// TIA Portal V20 export
FUNCTION_BLOCK "CallEquipment"   // FB17, LAD
TITLE = CallEquipment
AUTHOR : ERsystem_FA2_DH. Kim
// This block contains the logic and futher calls (e.g. sequences, control modules, diagnostics etc.) of the equipment module.
// stored: IsIECCheckEnabled true, MemoryReserve 100, Namespace Unit1.Em2, SetENOAutomatically false
   VAR_INPUT
      ZoneOperationEnable { ExternalWritable := 'False'} : "LWONIK_typeSafetyZoneManualOperation";
   END_VAR
   VAR_IN_OUT
      unitStatus : "LAF_typeUnitStatus";   // Current unit status o be used in this EM
      unitAlarmDB : "LAF_typeAlarms";   // Summarized EM Alarms for the Unit
      emFeedback : "LUC_typeEmFeedback";   // Feedback of the EM to the Unit
   END_VAR
   VAR
      instSequenceSemiAutoSplice { ExternalWritable := 'False'} : "Unit1.Em2.Sequence_1_SemiAutoSplice";   // EM Sequence Instance
      instHomeJob1 { S7_SetPoint := 'True'} : "LAF_SelectJob";
      instJob2 { S7_SetPoint := 'True'} : "LAF_SelectJob";
      instJob3 { S7_SetPoint := 'True'} : "LAF_SelectJob";
      instJob4 { S7_SetPoint := 'True'} : "LAF_SelectJob";
      instJob5 { S7_SetPoint := 'True'} : "LAF_SelectJob";
      instJob6 { S7_SetPoint := 'True'} : "LAF_SelectJob";
      instJob7 { S7_SetPoint := 'True'} : "LAF_SelectJob";
      instJob8 { S7_SetPoint := 'True'} : "LAF_SelectJob";
      instJob9 { S7_SetPoint := 'True'} : "LAF_SelectJob";
      instJob10 { S7_SetPoint := 'True'} : "LAF_SelectJob";
      instJob11 { S7_SetPoint := 'True'} : "LAF_SelectJob";
      instJob12 { S7_SetPoint := 'True'} : "LAF_SelectJob";
      instJob13 { S7_SetPoint := 'True'} : "LAF_SelectJob";
      instJob14 { S7_SetPoint := 'True'} : "LAF_SelectJob";
      instJob15 { S7_SetPoint := 'True'} : "LAF_SelectJob";
      instJob16 { S7_SetPoint := 'True'} : "LAF_SelectJob";
      instJob17 { S7_SetPoint := 'True'} : "LAF_SelectJob";
      instJob18 { S7_SetPoint := 'True'} : "LAF_SelectJob";
      instJob19 { S7_SetPoint := 'True'} : "LAF_SelectJob";
      instJob20 { S7_SetPoint := 'True'} : "LAF_SelectJob";
      instJob21 { S7_SetPoint := 'True'} : "LAF_SelectJob";
      instJob22 { S7_SetPoint := 'True'} : "LAF_SelectJob";
      instJob23 { S7_SetPoint := 'True'} : "LAF_SelectJob";
      instJob24 { S7_SetPoint := 'True'} : "LAF_SelectJob";
      instJob25 { S7_SetPoint := 'True'} : "LAF_SelectJob";
      instJob26 { S7_SetPoint := 'True'} : "LAF_SelectJob";
      instJob27 { S7_SetPoint := 'True'} : "LAF_SelectJob";
      instJob28 { S7_SetPoint := 'True'} : "LAF_SelectJob";
      instJob29 { S7_SetPoint := 'True'} : "LAF_SelectJob";
      instJob30 { S7_SetPoint := 'True'} : "LAF_SelectJob";
      instcmSuctionPadTopUpDown { ExternalAccessible := 'False'; ExternalVisible := 'False'; ExternalWritable := 'False'; S7_SetPoint := 'True'} : "LBC_TwoWayActuatorCn";
      instcmSuctionPadBtmUpDown { ExternalAccessible := 'False'; ExternalVisible := 'False'; ExternalWritable := 'False'; S7_SetPoint := 'True'} : "LBC_TwoWayActuatorCn";
      instcmCutterUpDown { ExternalAccessible := 'False'; ExternalVisible := 'False'; ExternalWritable := 'False'; S7_SetPoint := 'True'} : "LBC_TwoWayActuatorCn";
      instcmTapeTopUpDown { ExternalAccessible := 'False'; ExternalVisible := 'False'; ExternalWritable := 'False'; S7_SetPoint := 'True'} : "LBC_TwoWayActuatorCn";
      instcmTapeBtmUpDown { ExternalAccessible := 'False'; ExternalVisible := 'False'; ExternalWritable := 'False'; S7_SetPoint := 'True'} : "LBC_TwoWayActuatorCn";
      instcmSpliceHeadRotateTopFwdBwd { ExternalAccessible := 'False'; ExternalVisible := 'False'; ExternalWritable := 'False'; S7_SetPoint := 'True'} : "LBC_TwoWayActuatorCn";
      instcmSpliceHeadRotateBtmFwdBwd { ExternalAccessible := 'False'; ExternalVisible := 'False'; ExternalWritable := 'False'; S7_SetPoint := 'True'} : "LBC_TwoWayActuatorCn";
      instcmSuctionPadTopLeftVaccum { ExternalAccessible := 'False'; ExternalVisible := 'False'; ExternalWritable := 'False'; S7_SetPoint := 'True'} : "LBC_TwoWayActuatorCn";
      instcmSuctionPadTopRightVaccum { ExternalAccessible := 'False'; ExternalVisible := 'False'; ExternalWritable := 'False'; S7_SetPoint := 'True'} : "LBC_TwoWayActuatorCn";
      instCmSuctionPadBtmLeftVaccum { ExternalAccessible := 'False'; ExternalVisible := 'False'; ExternalWritable := 'False'; S7_SetPoint := 'True'} : "LBC_TwoWayActuatorCn";
      instCmSuctionPadBtmRightVaccum { ExternalAccessible := 'False'; ExternalVisible := 'False'; ExternalWritable := 'False'; S7_SetPoint := 'True'} : "LBC_TwoWayActuatorCn";
      instCmSuctionPadTopTapeVaccum { ExternalAccessible := 'False'; ExternalVisible := 'False'; ExternalWritable := 'False'; S7_SetPoint := 'True'} : "LBC_TwoWayActuatorCn";
      instCmSuctionPadBtmTapeVaccum { ExternalAccessible := 'False'; ExternalVisible := 'False'; ExternalWritable := 'False'; S7_SetPoint := 'True'} : "LBC_TwoWayActuatorCn";
      instManageAlarms { ExternalWritable := 'False'} : "LAF_ManageAlarms";
      instEventsPFE : "Unit1.Em2.EventsPFE";
      statTonTime { ExternalAccessible := 'False'; ExternalVisible := 'False'; ExternalWritable := 'False'} : Array[0..1999] of TON_TIME;
      statTofTime { ExternalAccessible := 'False'; ExternalVisible := 'False'; ExternalWritable := 'False'} : Array[0..99] of TOF_TIME;
      statPulse { ExternalAccessible := 'False'; ExternalVisible := 'False'; ExternalWritable := 'False'} : Array[0..999] of Bool;
      statUnitStatus { ExternalWritable := 'False'} : "LAF_typeUnitStatus";   // Unit Status used in this EM
      statEnableManualCmds : Bool;
      Scan_on { ExternalAccessible := 'False'; ExternalVisible := 'False'; ExternalWritable := 'False'} : Bool;
      "*** Interlock Actuator ******" { ExternalAccessible := 'False'; ExternalVisible := 'False'; ExternalWritable := 'False'; S7_SetPoint := 'True'} : Bool;
      "SuctionPadTopUpDown Home" { S7_SetPoint := 'True'} : "Cylinder.LER_Actuator";
      "SuctionPadTopUpDown Work" { S7_SetPoint := 'True'} : "Cylinder.LER_Actuator";
      "SuctionPadBtmUpDown Home" { S7_SetPoint := 'True'} : "Cylinder.LER_Actuator";
      "SuctionPadBtmUpDown Work" { S7_SetPoint := 'True'} : "Cylinder.LER_Actuator";
      "CutterUpDown Home" { S7_SetPoint := 'True'} : "Cylinder.LER_Actuator";
      "CutterUpDown Work" { S7_SetPoint := 'True'} : "Cylinder.LER_Actuator";
      "TapeTopUpDown Home" { S7_SetPoint := 'True'} : "Cylinder.LER_Actuator";
      "TapeTopUpDown Work" { S7_SetPoint := 'True'} : "Cylinder.LER_Actuator";
      "TapeBtmUpDown Home" { S7_SetPoint := 'True'} : "Cylinder.LER_Actuator";
      "TapeBtmUpDown Work" { S7_SetPoint := 'True'} : "Cylinder.LER_Actuator";
      "SpliceHeadRotateTopFwdBwd Home" { S7_SetPoint := 'True'} : "Cylinder.LER_Actuator";
      "SpliceHeadRotateTopFwdBwd Work" { S7_SetPoint := 'True'} : "Cylinder.LER_Actuator";
      "SpliceHeadRotateBtmFwdBwd Home" { S7_SetPoint := 'True'} : "Cylinder.LER_Actuator";
      "SpliceHeadRotateBtmFwdBwd Work" { S7_SetPoint := 'True'} : "Cylinder.LER_Actuator";
      Cylinder3 : "LER_CM_Name";
      Vaccum1 : "LER_CM_Name";
      Vaccum6 : "LER_CM_Name";
      Cylinder8 : "LER_CM_Name";
      citi_Ptrig : Array[0..20] of Bool;
      citiTon : Array[0..20] of TON_TIME;
      citi : Time;
      citiTest : Array[0..20] of Bool;
   END_VAR
   VAR_TEMP
      tempScInProduction : Bool;   // Mode Production and StateComplete
      tempScNoProduction : Bool;   // Mode Manual and StateComplete
   END_VAR
   VAR CONSTANT
      delayTime : Time := T#3s;
      TRUE : Bool := TRUE;   // Template : Add em specific conditions here
      FALSE : Bool := FALSE;
      NO_JOB : DInt;   // No job
      MIN_POSITION_NUMBER : SInt;
      INIT_POSITION_NUMBER : SInt := -1;
   END_VAR
   VAR_TEMP   // added for the SCL form of the ladder/FBD networks
      _w1 : Bool;
      _w2 : Bool;
      _w3 : Bool;
      _w4 : Bool;
      _w5 : Bool;
      _w6 : Bool;
      _w7 : Bool;
      _w8 : Bool;
      _w9 : Bool;
      _w10 : Bool;
      _w11 : Bool;
      _w12 : Bool;
      _w13 : Bool;
      _w14 : Bool;
      _w15 : Bool;
      _w16 : Bool;
      _w17 : Bool;
      _w18 : Bool;
      _w19 : Bool;
      _w20 : Bool;
   END_VAR
BEGIN

REGION Network 1: BLOCK INFO HEADER
   // (company) / (C) Copyright (year)
   // ---------------------------------------------------------------------------------
   // Title:                             (Title of this block)
   // Comment/Function: (that is implemented in the block)
   // Library/Family:           (that the source is dedicated to)
   // Author:                        (department / person in charge / contact)
   // Target System:          (test system with FW version)
   // Engineering:              TIA Portal (SW version)
   // Restrictions:               (OB types, etc.)
   // Requirements:           (hardware, technological package, etc.)
   // ---------------------------------------------------------------------------------
   // Change log table:
   // Version          | Date             | Signature      | Expert in charge  | Changes applied ------------------------|----------------------|-------------------------|--------------------------------|-----------------------
   // 001.000.000 | yyyy-mm-dd | 0x00000000 | (name of expert) | First released version
END_REGION

REGION Network 2: DESCRIPTION
   // This is a template block provided by the Automation Framework. It can be used to create an own project.
   // The Block Info Header is prepared to put in your own data.
   // Description of the block could be added here and the docu created by Code2Docu.
END_REGION

REGION Network 3: disableFeedbackHomePos
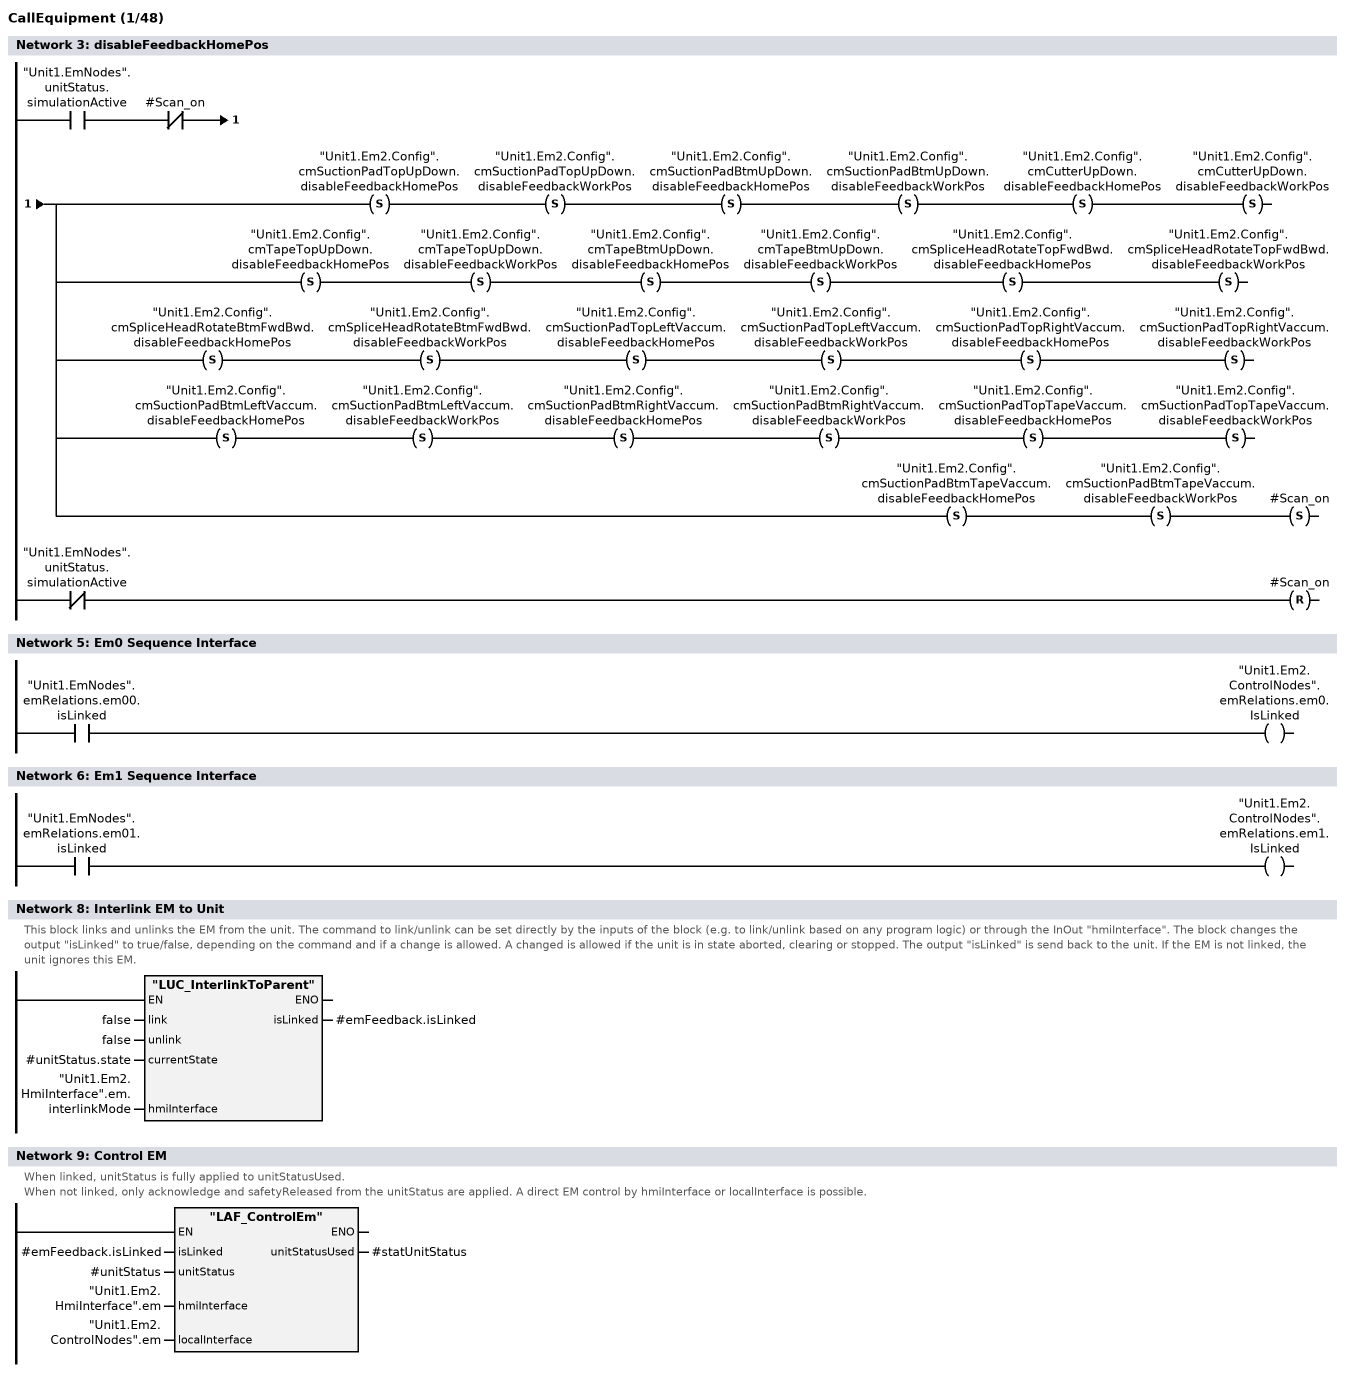
   RUNG wire#powerrail
      Contact( "Unit1.EmNodes".unitStatus.simulationActive )
      I_Contact( #Scan_on )
      wire#w1
      S_Coil( "Unit1.Em2.Config".cmSuctionPadTopUpDown.disableFeedbackHomePos )
      S_Coil( "Unit1.Em2.Config".cmSuctionPadTopUpDown.disableFeedbackWorkPos )
      S_Coil( "Unit1.Em2.Config".cmSuctionPadBtmUpDown.disableFeedbackHomePos )
      S_Coil( "Unit1.Em2.Config".cmSuctionPadBtmUpDown.disableFeedbackWorkPos )
      S_Coil( "Unit1.Em2.Config".cmCutterUpDown.disableFeedbackHomePos )
      S_Coil( "Unit1.Em2.Config".cmCutterUpDown.disableFeedbackWorkPos )
   END_RUNG
   RUNG wire#w1
      S_Coil( "Unit1.Em2.Config".cmTapeTopUpDown.disableFeedbackHomePos )
      S_Coil( "Unit1.Em2.Config".cmTapeTopUpDown.disableFeedbackWorkPos )
      S_Coil( "Unit1.Em2.Config".cmTapeBtmUpDown.disableFeedbackHomePos )
      S_Coil( "Unit1.Em2.Config".cmTapeBtmUpDown.disableFeedbackWorkPos )
      S_Coil( "Unit1.Em2.Config".cmSpliceHeadRotateTopFwdBwd.disableFeedbackHomePos )
      S_Coil( "Unit1.Em2.Config".cmSpliceHeadRotateTopFwdBwd.disableFeedbackWorkPos )
   END_RUNG
   RUNG wire#w1
      S_Coil( "Unit1.Em2.Config".cmSpliceHeadRotateBtmFwdBwd.disableFeedbackHomePos )
      S_Coil( "Unit1.Em2.Config".cmSpliceHeadRotateBtmFwdBwd.disableFeedbackWorkPos )
      S_Coil( "Unit1.Em2.Config".cmSuctionPadTopLeftVaccum.disableFeedbackHomePos )
      S_Coil( "Unit1.Em2.Config".cmSuctionPadTopLeftVaccum.disableFeedbackWorkPos )
      S_Coil( "Unit1.Em2.Config".cmSuctionPadTopRightVaccum.disableFeedbackHomePos )
      S_Coil( "Unit1.Em2.Config".cmSuctionPadTopRightVaccum.disableFeedbackWorkPos )
   END_RUNG
   RUNG wire#w1
      S_Coil( "Unit1.Em2.Config".cmSuctionPadBtmLeftVaccum.disableFeedbackHomePos )
      S_Coil( "Unit1.Em2.Config".cmSuctionPadBtmLeftVaccum.disableFeedbackWorkPos )
      S_Coil( "Unit1.Em2.Config".cmSuctionPadBtmRightVaccum.disableFeedbackHomePos )
      S_Coil( "Unit1.Em2.Config".cmSuctionPadBtmRightVaccum.disableFeedbackWorkPos )
      S_Coil( "Unit1.Em2.Config".cmSuctionPadTopTapeVaccum.disableFeedbackHomePos )
      S_Coil( "Unit1.Em2.Config".cmSuctionPadTopTapeVaccum.disableFeedbackWorkPos )
   END_RUNG
   RUNG wire#w1
      S_Coil( "Unit1.Em2.Config".cmSuctionPadBtmTapeVaccum.disableFeedbackHomePos )
      S_Coil( "Unit1.Em2.Config".cmSuctionPadBtmTapeVaccum.disableFeedbackWorkPos )
      S_Coil( #Scan_on )
   END_RUNG
   RUNG wire#powerrail
      I_Contact( "Unit1.EmNodes".unitStatus.simulationActive )
      R_Coil( #Scan_on )
   END_RUNG
   // the same network as SCL:
   IF "Unit1.EmNodes".unitStatus.simulationActive AND NOT #Scan_on THEN
       "Unit1.Em2.Config".cmSuctionPadTopUpDown.disableFeedbackHomePos := TRUE;
       "Unit1.Em2.Config".cmSuctionPadTopUpDown.disableFeedbackWorkPos := TRUE;
       "Unit1.Em2.Config".cmSuctionPadBtmUpDown.disableFeedbackHomePos := TRUE;
       "Unit1.Em2.Config".cmSuctionPadBtmUpDown.disableFeedbackWorkPos := TRUE;
       "Unit1.Em2.Config".cmCutterUpDown.disableFeedbackHomePos := TRUE;
       "Unit1.Em2.Config".cmCutterUpDown.disableFeedbackWorkPos := TRUE;
       "Unit1.Em2.Config".cmTapeTopUpDown.disableFeedbackHomePos := TRUE;
       "Unit1.Em2.Config".cmTapeTopUpDown.disableFeedbackWorkPos := TRUE;
       "Unit1.Em2.Config".cmTapeBtmUpDown.disableFeedbackHomePos := TRUE;
       "Unit1.Em2.Config".cmTapeBtmUpDown.disableFeedbackWorkPos := TRUE;
       "Unit1.Em2.Config".cmSpliceHeadRotateTopFwdBwd.disableFeedbackHomePos := TRUE;
       "Unit1.Em2.Config".cmSpliceHeadRotateTopFwdBwd.disableFeedbackWorkPos := TRUE;
       "Unit1.Em2.Config".cmSpliceHeadRotateBtmFwdBwd.disableFeedbackHomePos := TRUE;
       "Unit1.Em2.Config".cmSpliceHeadRotateBtmFwdBwd.disableFeedbackWorkPos := TRUE;
       "Unit1.Em2.Config".cmSuctionPadTopLeftVaccum.disableFeedbackHomePos := TRUE;
       "Unit1.Em2.Config".cmSuctionPadTopLeftVaccum.disableFeedbackWorkPos := TRUE;
       "Unit1.Em2.Config".cmSuctionPadTopRightVaccum.disableFeedbackHomePos := TRUE;
       "Unit1.Em2.Config".cmSuctionPadTopRightVaccum.disableFeedbackWorkPos := TRUE;
       "Unit1.Em2.Config".cmSuctionPadBtmLeftVaccum.disableFeedbackHomePos := TRUE;
       "Unit1.Em2.Config".cmSuctionPadBtmLeftVaccum.disableFeedbackWorkPos := TRUE;
       "Unit1.Em2.Config".cmSuctionPadBtmRightVaccum.disableFeedbackHomePos := TRUE;
       "Unit1.Em2.Config".cmSuctionPadBtmRightVaccum.disableFeedbackWorkPos := TRUE;
       "Unit1.Em2.Config".cmSuctionPadTopTapeVaccum.disableFeedbackHomePos := TRUE;
       "Unit1.Em2.Config".cmSuctionPadTopTapeVaccum.disableFeedbackWorkPos := TRUE;
       "Unit1.Em2.Config".cmSuctionPadBtmTapeVaccum.disableFeedbackHomePos := TRUE;
       "Unit1.Em2.Config".cmSuctionPadBtmTapeVaccum.disableFeedbackWorkPos := TRUE;
       #Scan_on := TRUE;
   END_IF;
   IF NOT "Unit1.EmNodes".unitStatus.simulationActive THEN #Scan_on := FALSE; END_IF;
END_REGION

REGION Network 4: ******************** Unit Input ********************
END_REGION

REGION Network 5: Em0 Sequence Interface
   RUNG wire#powerrail
      Contact( "Unit1.EmNodes".emRelations.em00.isLinked )
      Coil( "Unit1.Em2.ControlNodes".emRelations.em0.IsLinked )
   END_RUNG
   // the same network as SCL:
   "Unit1.Em2.ControlNodes".emRelations.em0.IsLinked := "Unit1.EmNodes".emRelations.em00.isLinked;
END_REGION

REGION Network 6: Em1 Sequence Interface
   RUNG wire#powerrail
      Contact( "Unit1.EmNodes".emRelations.em01.isLinked )
      Coil( "Unit1.Em2.ControlNodes".emRelations.em1.IsLinked )
   END_RUNG
   // the same network as SCL:
   "Unit1.Em2.ControlNodes".emRelations.em1.IsLinked := "Unit1.EmNodes".emRelations.em01.isLinked;
END_REGION

REGION Network 7: *************** Equipment Control **************************
END_REGION

REGION Network 8: Interlink EM to Unit
   // This block links and unlinks the EM from the unit. The command to link/unlink can be set directly by the inputs of the block (e.g. to link/unlink based on any program logic) or through the InOut "hmiInterface". The block changes the output "isLinked" to true/false, depending on the command and if a change is allowed. A changed is allowed if the unit is in state aborted, clearing or stopped. The output "isLinked" is send back to the unit. If the EM is not linked, the unit ignores this EM.
   RUNG wire#powerrail
      "LUC_InterlinkToParent"(link := false, unlink := false, currentState := #unitStatus.state, hmiInterface := "Unit1.Em2.HmiInterface".em.interlinkMode, isLinked => #emFeedback.isLinked)
   END_RUNG
   // the same network as SCL:
   "LUC_InterlinkToParent"(link := false,
                           unlink := false,
                           currentState := #unitStatus.state,
                           hmiInterface := "Unit1.Em2.HmiInterface".em.interlinkMode,
                           isLinked => #emFeedback.isLinked);
END_REGION

REGION Network 9: Control EM
   // When linked, unitStatus is fully applied to unitStatusUsed.
   // When not linked, only acknowledge and safetyReleased from the unitStatus are applied. A direct EM control by hmiInterface or localInterface is possible.
   RUNG wire#powerrail
      "LAF_ControlEm"(isLinked := #emFeedback.isLinked, unitStatus := #unitStatus, hmiInterface := "Unit1.Em2.HmiInterface".em, localInterface := "Unit1.Em2.ControlNodes".em, unitStatusUsed => #statUnitStatus)
   END_RUNG
   // the same network as SCL:
   "LAF_ControlEm"(isLinked := #emFeedback.isLinked,
                   unitStatus := #unitStatus,
                   hmiInterface := "Unit1.Em2.HmiInterface".em,
                   localInterface := "Unit1.Em2.ControlNodes".em,
                   unitStatusUsed => #statUnitStatus);
END_REGION

REGION Network 10: EnableManualCmds
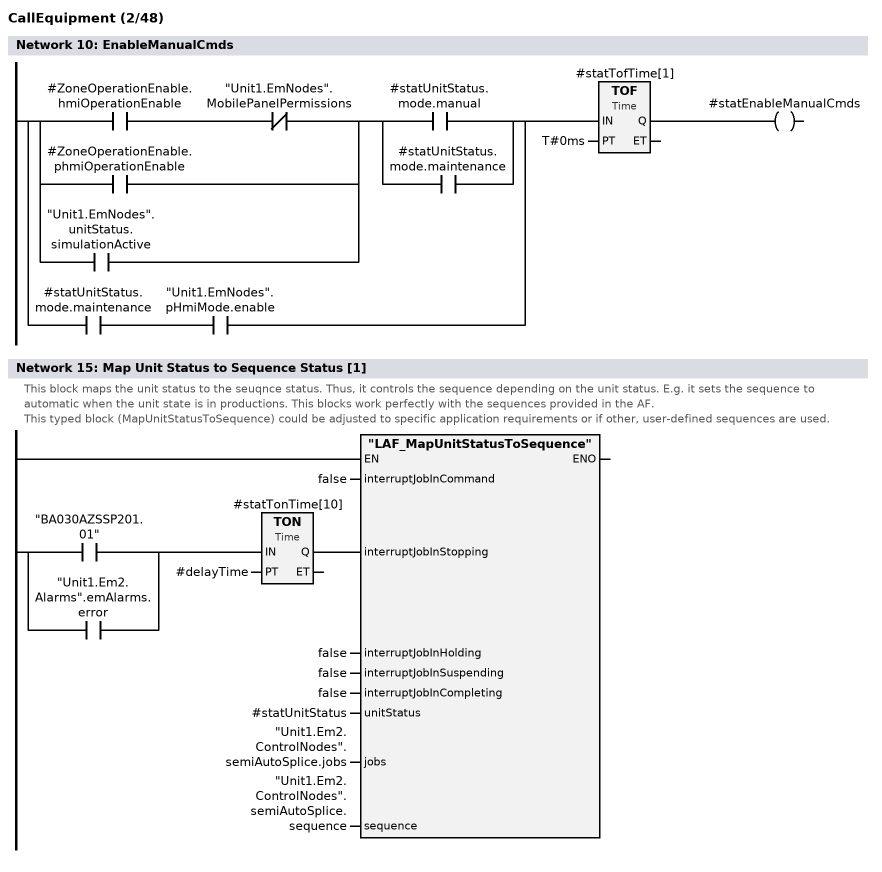
   RUNG wire#powerrail
      Contact( #ZoneOperationEnable.hmiOperationEnable )
      I_Contact( "Unit1.EmNodes".MobilePanelPermissions )
      wire#w1
      Contact( #statUnitStatus.mode.manual )
      wire#w2
      { S7_Templates := "time_type := Time" } #statTofTime[1].TOF(pt := T#0ms, et =>)
      Coil( #statEnableManualCmds )
   END_RUNG
   RUNG wire#powerrail
      Contact( #ZoneOperationEnable.phmiOperationEnable )
   END_RUNG wire#w1
   RUNG wire#powerrail
      Contact( "Unit1.EmNodes".unitStatus.simulationActive )
   END_RUNG wire#w1
   RUNG wire#w1
      Contact( #statUnitStatus.mode.maintenance )
   END_RUNG wire#w2
   RUNG wire#powerrail
      Contact( #statUnitStatus.mode.maintenance )
      Contact( "Unit1.EmNodes".pHmiMode.enable )
   END_RUNG wire#w2
   // the same network as SCL:
   #statTofTime[1].TOF(IN := (((#ZoneOperationEnable.hmiOperationEnable AND NOT "Unit1.EmNodes".MobilePanelPermissions) OR #ZoneOperationEnable.phmiOperationEnable OR "Unit1.EmNodes".unitStatus.simulationActive) AND (#statUnitStatus.mode.manual OR #statUnitStatus.mode.maintenance)) OR (#statUnitStatus.mode.maintenance AND "Unit1.EmNodes".pHmiMode.enable),
                       PT := T#0ms);
   #statEnableManualCmds := #statTofTime[1].Q;
END_REGION

REGION Network 12: *************** Control Modules (Sensors) ********************
   // Call control modules that are sensors before the em logic (jobs and sequence), so that the latest value is used in the logic.
END_REGION

REGION Network 14: *************** Equipment Logic ***************************
END_REGION

REGION Network 15: Map Unit Status to Sequence Status [1]
   // This block maps the unit status to the seuqnce status. Thus, it controls the sequence depending on the unit status. E.g. it sets the sequence to automatic when the unit state is in productions. This blocks work perfectly with the sequences provided in the AF. 
   // This typed block (MapUnitStatusToSequence) could be adjusted to specific application requirements or if other, user-defined sequences are used.
   RUNG wire#powerrail
      "LAF_MapUnitStatusToSequence"(interruptJobInStopping := wire#w2, interruptJobInCommand := false, interruptJobInHolding := false, interruptJobInSuspending := false, interruptJobInCompleting := false, unitStatus := #statUnitStatus, jobs := "Unit1.Em2.ControlNodes".semiAutoSplice.jobs, sequence := "Unit1.Em2.ControlNodes".semiAutoSplice.sequence)
   END_RUNG
   RUNG wire#powerrail
      Contact( "BA030AZSSP201.01" )
      wire#w1
      { S7_Templates := "time_type := Time" } #statTonTime[10].TON(pt := #delayTime, et =>)
   END_RUNG wire#w2
   RUNG wire#powerrail
      Contact( "Unit1.Em2.Alarms".emAlarms.error )
   END_RUNG wire#w1
   // the same network as SCL:
   #statTonTime[10].TON(IN := "BA030AZSSP201.01" OR "Unit1.Em2.Alarms".emAlarms.error, PT := #delayTime);
   "LAF_MapUnitStatusToSequence"(interruptJobInCommand := false,
                           interruptJobInStopping := #statTonTime[10].Q,
                           interruptJobInHolding := false,
                           interruptJobInSuspending := false,
                           interruptJobInCompleting := false,
                           unitStatus := #statUnitStatus,
                           jobs := "Unit1.Em2.ControlNodes".semiAutoSplice.jobs,
                           sequence := "Unit1.Em2.ControlNodes".semiAutoSplice.sequence);
END_REGION

REGION Network 17: Select Job [1] Tape Unit Initialized
   // Decide which Step Sequence to start depending on the OMAC State and EM conditions
   // First Move Block is to Initialize the jobSelect Number
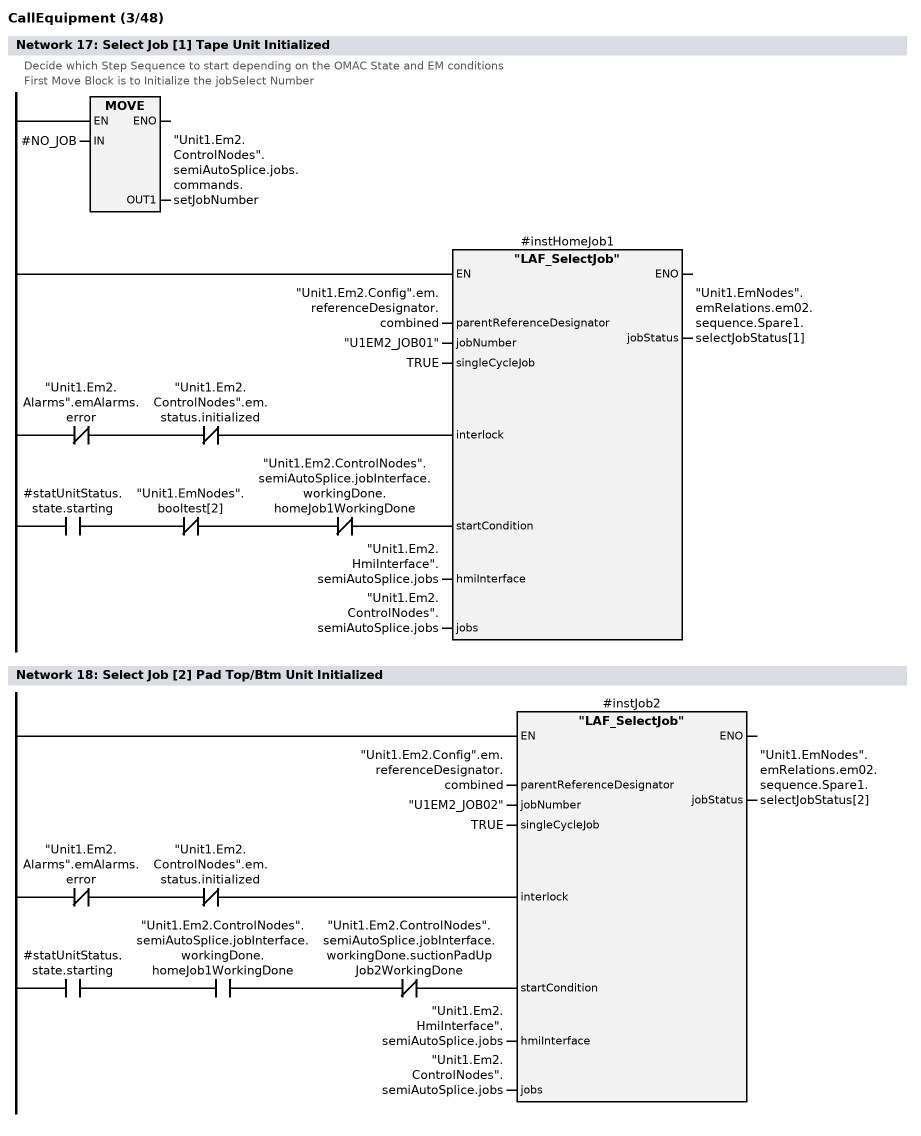
   RUNG wire#powerrail
      Move(in := #NO_JOB, out1 => "Unit1.Em2.ControlNodes".semiAutoSplice.jobs.commands.setJobNumber)
   END_RUNG
   RUNG wire#powerrail
      #instHomeJob1(interlock := wire#w1, startCondition := wire#w2, parentReferenceDesignator := "Unit1.Em2.Config".em.referenceDesignator.combined, jobNumber := "U1EM2_JOB01", singleCycleJob := TRUE, hmiInterface := "Unit1.Em2.HmiInterface".semiAutoSplice.jobs, jobs := "Unit1.Em2.ControlNodes".semiAutoSplice.jobs, jobStatus => "Unit1.EmNodes".emRelations.em02.sequence.Spare1.selectJobStatus[1])
   END_RUNG
   RUNG wire#powerrail
      I_Contact( "Unit1.Em2.Alarms".emAlarms.error )
      I_Contact( "Unit1.Em2.ControlNodes".em.status.initialized )
   END_RUNG wire#w1
   RUNG wire#powerrail
      Contact( #statUnitStatus.state.starting )
      I_Contact( "Unit1.EmNodes".booltest[2] )
      I_Contact( "Unit1.Em2.ControlNodes".semiAutoSplice.jobInterface.workingDone.homeJob1WorkingDone )
   END_RUNG wire#w2
   // the same network as SCL:
   "Unit1.Em2.ControlNodes".semiAutoSplice.jobs.commands.setJobNumber := #NO_JOB;
   #instHomeJob1(parentReferenceDesignator := "Unit1.Em2.Config".em.referenceDesignator.combined,   // "LAF_SelectJob"
                 jobNumber := "U1EM2_JOB01",
                 singleCycleJob := TRUE,
                 interlock := NOT "Unit1.Em2.Alarms".emAlarms.error AND NOT "Unit1.Em2.ControlNodes".em.status.initialized,
                 startCondition := #statUnitStatus.state.starting AND NOT "Unit1.EmNodes".booltest[2] AND NOT "Unit1.Em2.ControlNodes".semiAutoSplice.jobInterface.workingDone.homeJob1WorkingDone,
                 hmiInterface := "Unit1.Em2.HmiInterface".semiAutoSplice.jobs,
                 jobs := "Unit1.Em2.ControlNodes".semiAutoSplice.jobs,
                 jobStatus => "Unit1.EmNodes".emRelations.em02.sequence.Spare1.selectJobStatus[1]);
END_REGION

REGION Network 18: Select Job [2] Pad Top/Btm Unit Initialized
   RUNG wire#powerrail
      #instJob2(interlock := wire#w1, startCondition := wire#w2, parentReferenceDesignator := "Unit1.Em2.Config".em.referenceDesignator.combined, jobNumber := "U1EM2_JOB02", singleCycleJob := TRUE, hmiInterface := "Unit1.Em2.HmiInterface".semiAutoSplice.jobs, jobs := "Unit1.Em2.ControlNodes".semiAutoSplice.jobs, jobStatus => "Unit1.EmNodes".emRelations.em02.sequence.Spare1.selectJobStatus[2])
   END_RUNG
   RUNG wire#powerrail
      I_Contact( "Unit1.Em2.Alarms".emAlarms.error )
      I_Contact( "Unit1.Em2.ControlNodes".em.status.initialized )
   END_RUNG wire#w1
   RUNG wire#powerrail
      Contact( #statUnitStatus.state.starting )
      Contact( "Unit1.Em2.ControlNodes".semiAutoSplice.jobInterface.workingDone.homeJob1WorkingDone )
      I_Contact( "Unit1.Em2.ControlNodes".semiAutoSplice.jobInterface.workingDone.suctionPadUpJob2WorkingDone )
   END_RUNG wire#w2
   // the same network as SCL:
   #instJob2(parentReferenceDesignator := "Unit1.Em2.Config".em.referenceDesignator.combined,   // "LAF_SelectJob"
             jobNumber := "U1EM2_JOB02",
             singleCycleJob := TRUE,
             interlock := NOT "Unit1.Em2.Alarms".emAlarms.error AND NOT "Unit1.Em2.ControlNodes".em.status.initialized,
             startCondition := #statUnitStatus.state.starting AND "Unit1.Em2.ControlNodes".semiAutoSplice.jobInterface.workingDone.homeJob1WorkingDone AND NOT "Unit1.Em2.ControlNodes".semiAutoSplice.jobInterface.workingDone.suctionPadUpJob2WorkingDone,
             hmiInterface := "Unit1.Em2.HmiInterface".semiAutoSplice.jobs,
             jobs := "Unit1.Em2.ControlNodes".semiAutoSplice.jobs,
             jobStatus => "Unit1.EmNodes".emRelations.em02.sequence.Spare1.selectJobStatus[2]);
END_REGION

REGION Network 19: Select Job [3] Head Rotate Top/Btm Unit Initialized
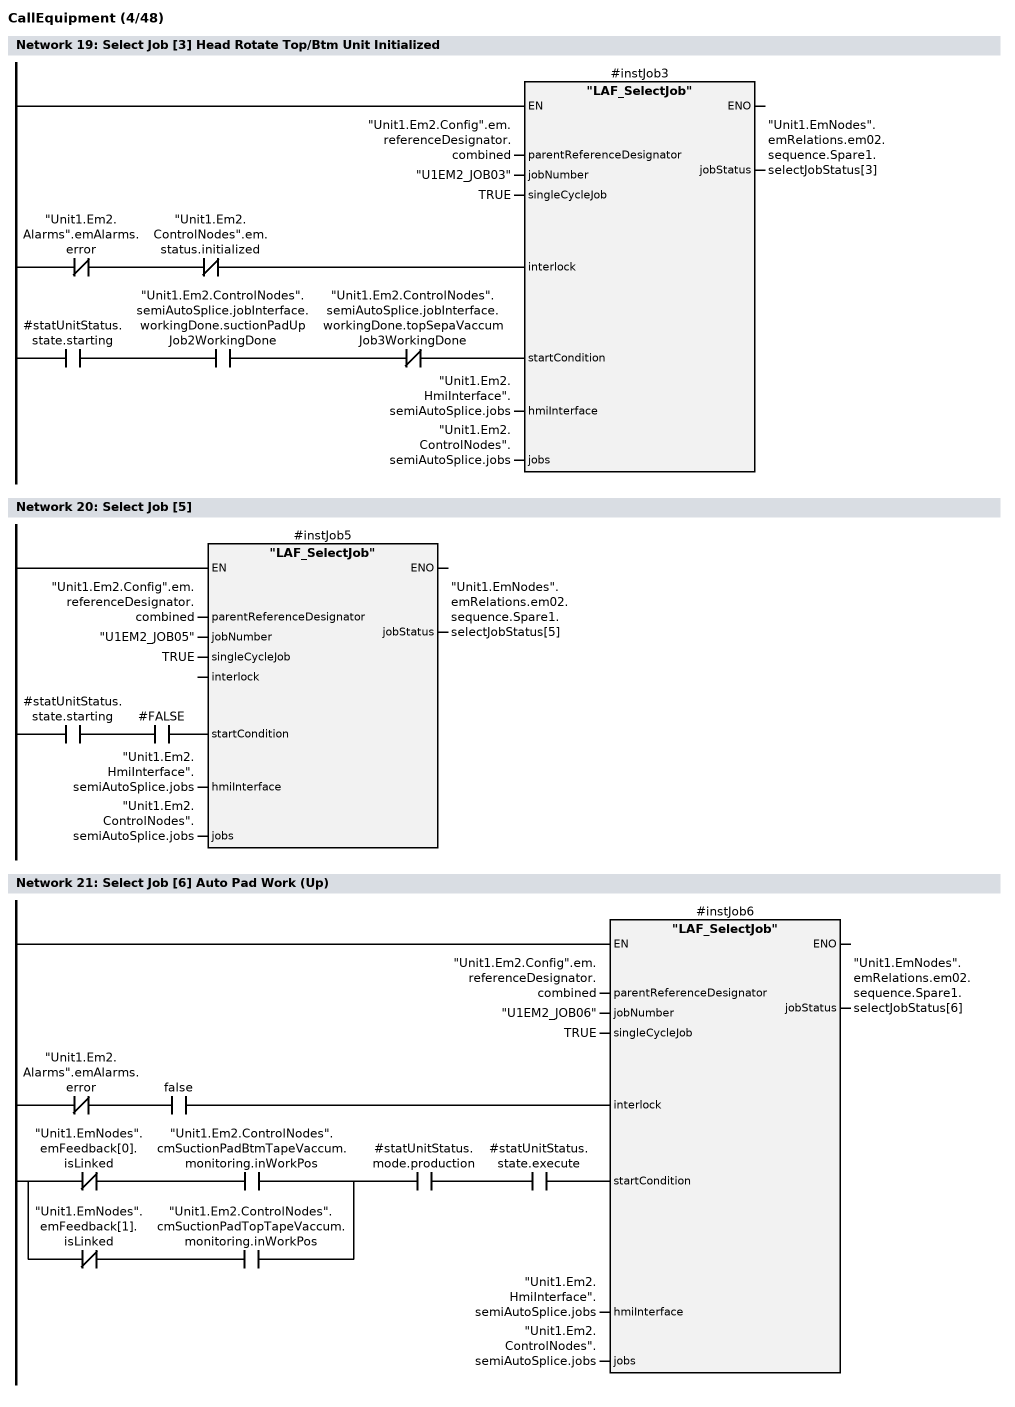
   RUNG wire#powerrail
      #instJob3(interlock := wire#w1, startCondition := wire#w2, parentReferenceDesignator := "Unit1.Em2.Config".em.referenceDesignator.combined, jobNumber := "U1EM2_JOB03", singleCycleJob := TRUE, hmiInterface := "Unit1.Em2.HmiInterface".semiAutoSplice.jobs, jobs := "Unit1.Em2.ControlNodes".semiAutoSplice.jobs, jobStatus => "Unit1.EmNodes".emRelations.em02.sequence.Spare1.selectJobStatus[3])
   END_RUNG
   RUNG wire#powerrail
      I_Contact( "Unit1.Em2.Alarms".emAlarms.error )
      I_Contact( "Unit1.Em2.ControlNodes".em.status.initialized )
   END_RUNG wire#w1
   RUNG wire#powerrail
      Contact( #statUnitStatus.state.starting )
      Contact( "Unit1.Em2.ControlNodes".semiAutoSplice.jobInterface.workingDone.suctionPadUpJob2WorkingDone )
      I_Contact( "Unit1.Em2.ControlNodes".semiAutoSplice.jobInterface.workingDone.topSepaVaccumJob3WorkingDone )
   END_RUNG wire#w2
   // the same network as SCL:
   #instJob3(parentReferenceDesignator := "Unit1.Em2.Config".em.referenceDesignator.combined,   // "LAF_SelectJob"
             jobNumber := "U1EM2_JOB03",
             singleCycleJob := TRUE,
             interlock := NOT "Unit1.Em2.Alarms".emAlarms.error AND NOT "Unit1.Em2.ControlNodes".em.status.initialized,
             startCondition := #statUnitStatus.state.starting AND "Unit1.Em2.ControlNodes".semiAutoSplice.jobInterface.workingDone.suctionPadUpJob2WorkingDone AND NOT "Unit1.Em2.ControlNodes".semiAutoSplice.jobInterface.workingDone.topSepaVaccumJob3WorkingDone,
             hmiInterface := "Unit1.Em2.HmiInterface".semiAutoSplice.jobs,
             jobs := "Unit1.Em2.ControlNodes".semiAutoSplice.jobs,
             jobStatus => "Unit1.EmNodes".emRelations.em02.sequence.Spare1.selectJobStatus[3]);
END_REGION

REGION Network 20: Select Job [5]
   RUNG wire#powerrail
      #instJob5(startCondition := wire#w1, parentReferenceDesignator := "Unit1.Em2.Config".em.referenceDesignator.combined, jobNumber := "U1EM2_JOB05", singleCycleJob := TRUE, interlock :=, hmiInterface := "Unit1.Em2.HmiInterface".semiAutoSplice.jobs, jobs := "Unit1.Em2.ControlNodes".semiAutoSplice.jobs, jobStatus => "Unit1.EmNodes".emRelations.em02.sequence.Spare1.selectJobStatus[5])
   END_RUNG
   RUNG wire#powerrail
      Contact( #statUnitStatus.state.starting )
      Contact( #FALSE )
   END_RUNG wire#w1
   // the same network as SCL:
   #instJob5(parentReferenceDesignator := "Unit1.Em2.Config".em.referenceDesignator.combined,   // "LAF_SelectJob"
             jobNumber := "U1EM2_JOB05",
             singleCycleJob := TRUE,
             startCondition := #statUnitStatus.state.starting AND #FALSE,
             hmiInterface := "Unit1.Em2.HmiInterface".semiAutoSplice.jobs,
             jobs := "Unit1.Em2.ControlNodes".semiAutoSplice.jobs,
             jobStatus => "Unit1.EmNodes".emRelations.em02.sequence.Spare1.selectJobStatus[5]);
END_REGION

REGION Network 21: Select Job [6] Auto Pad Work (Up)
   RUNG wire#powerrail
      #instJob6(interlock := wire#w1, startCondition := wire#w3, parentReferenceDesignator := "Unit1.Em2.Config".em.referenceDesignator.combined, jobNumber := "U1EM2_JOB06", singleCycleJob := TRUE, hmiInterface := "Unit1.Em2.HmiInterface".semiAutoSplice.jobs, jobs := "Unit1.Em2.ControlNodes".semiAutoSplice.jobs, jobStatus => "Unit1.EmNodes".emRelations.em02.sequence.Spare1.selectJobStatus[6])
   END_RUNG
   RUNG wire#powerrail
      I_Contact( "Unit1.Em2.Alarms".emAlarms.error )
      Contact( false )
   END_RUNG wire#w1
   RUNG wire#powerrail
      I_Contact( "Unit1.EmNodes".emFeedback[0].isLinked )
      Contact( "Unit1.Em2.ControlNodes".cmSuctionPadBtmTapeVaccum.monitoring.inWorkPos )
      wire#w2
      Contact( #statUnitStatus.mode.production )
      Contact( #statUnitStatus.state.execute )
   END_RUNG wire#w3
   RUNG wire#powerrail
      I_Contact( "Unit1.EmNodes".emFeedback[1].isLinked )
      Contact( "Unit1.Em2.ControlNodes".cmSuctionPadTopTapeVaccum.monitoring.inWorkPos )
   END_RUNG wire#w2
   // the same network as SCL:
   #instJob6(parentReferenceDesignator := "Unit1.Em2.Config".em.referenceDesignator.combined,   // "LAF_SelectJob"
             jobNumber := "U1EM2_JOB06",
             singleCycleJob := TRUE,
             interlock := NOT "Unit1.Em2.Alarms".emAlarms.error AND false,
             startCondition := ((NOT "Unit1.EmNodes".emFeedback[0].isLinked AND "Unit1.Em2.ControlNodes".cmSuctionPadBtmTapeVaccum.monitoring.inWorkPos) OR (NOT "Unit1.EmNodes".emFeedback[1].isLinked AND "Unit1.Em2.ControlNodes".cmSuctionPadTopTapeVaccum.monitoring.inWorkPos)) AND #statUnitStatus.mode.production AND #statUnitStatus.state.execute,
             hmiInterface := "Unit1.Em2.HmiInterface".semiAutoSplice.jobs,
             jobs := "Unit1.Em2.ControlNodes".semiAutoSplice.jobs,
             jobStatus => "Unit1.EmNodes".emRelations.em02.sequence.Spare1.selectJobStatus[6]);
END_REGION

REGION Network 22: Select Job [7] Auto Suction Pad Vaccum
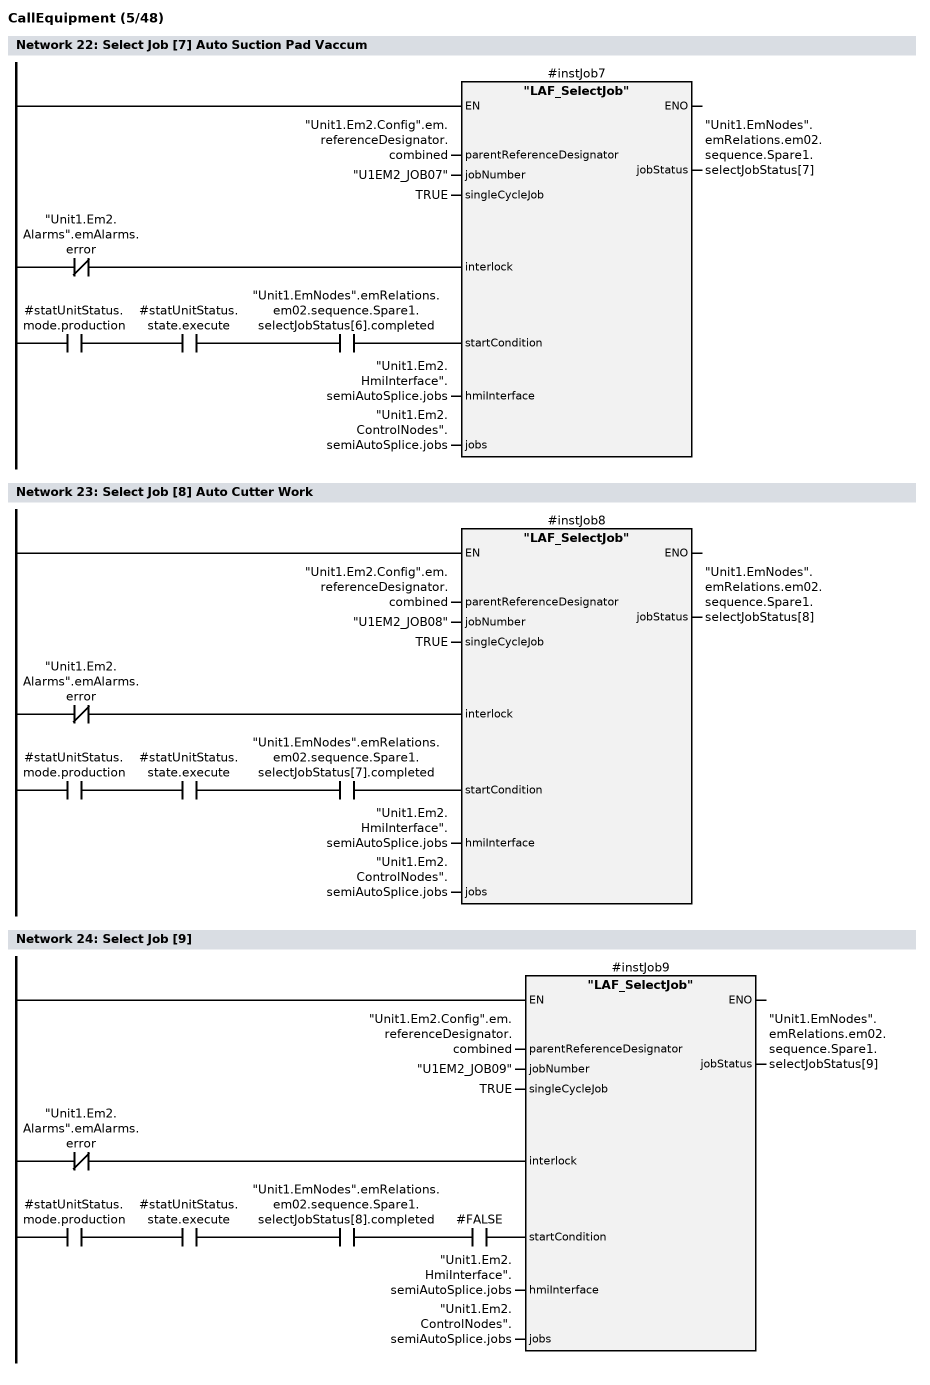
   RUNG wire#powerrail
      #instJob7(interlock := wire#w1, startCondition := wire#w2, parentReferenceDesignator := "Unit1.Em2.Config".em.referenceDesignator.combined, jobNumber := "U1EM2_JOB07", singleCycleJob := TRUE, hmiInterface := "Unit1.Em2.HmiInterface".semiAutoSplice.jobs, jobs := "Unit1.Em2.ControlNodes".semiAutoSplice.jobs, jobStatus => "Unit1.EmNodes".emRelations.em02.sequence.Spare1.selectJobStatus[7])
   END_RUNG
   RUNG wire#powerrail
      I_Contact( "Unit1.Em2.Alarms".emAlarms.error )
   END_RUNG wire#w1
   RUNG wire#powerrail
      Contact( #statUnitStatus.mode.production )
      Contact( #statUnitStatus.state.execute )
      Contact( "Unit1.EmNodes".emRelations.em02.sequence.Spare1.selectJobStatus[6].completed )
   END_RUNG wire#w2
   // the same network as SCL:
   #instJob7(parentReferenceDesignator := "Unit1.Em2.Config".em.referenceDesignator.combined,   // "LAF_SelectJob"
             jobNumber := "U1EM2_JOB07",
             singleCycleJob := TRUE,
             interlock := NOT "Unit1.Em2.Alarms".emAlarms.error,
             startCondition := #statUnitStatus.mode.production AND #statUnitStatus.state.execute AND "Unit1.EmNodes".emRelations.em02.sequence.Spare1.selectJobStatus[6].completed,
             hmiInterface := "Unit1.Em2.HmiInterface".semiAutoSplice.jobs,
             jobs := "Unit1.Em2.ControlNodes".semiAutoSplice.jobs,
             jobStatus => "Unit1.EmNodes".emRelations.em02.sequence.Spare1.selectJobStatus[7]);
END_REGION

REGION Network 23: Select Job [8] Auto Cutter Work
   RUNG wire#powerrail
      #instJob8(interlock := wire#w1, startCondition := wire#w2, parentReferenceDesignator := "Unit1.Em2.Config".em.referenceDesignator.combined, jobNumber := "U1EM2_JOB08", singleCycleJob := TRUE, hmiInterface := "Unit1.Em2.HmiInterface".semiAutoSplice.jobs, jobs := "Unit1.Em2.ControlNodes".semiAutoSplice.jobs, jobStatus => "Unit1.EmNodes".emRelations.em02.sequence.Spare1.selectJobStatus[8])
   END_RUNG
   RUNG wire#powerrail
      I_Contact( "Unit1.Em2.Alarms".emAlarms.error )
   END_RUNG wire#w1
   RUNG wire#powerrail
      Contact( #statUnitStatus.mode.production )
      Contact( #statUnitStatus.state.execute )
      Contact( "Unit1.EmNodes".emRelations.em02.sequence.Spare1.selectJobStatus[7].completed )
   END_RUNG wire#w2
   // the same network as SCL:
   #instJob8(parentReferenceDesignator := "Unit1.Em2.Config".em.referenceDesignator.combined,   // "LAF_SelectJob"
             jobNumber := "U1EM2_JOB08",
             singleCycleJob := TRUE,
             interlock := NOT "Unit1.Em2.Alarms".emAlarms.error,
             startCondition := #statUnitStatus.mode.production AND #statUnitStatus.state.execute AND "Unit1.EmNodes".emRelations.em02.sequence.Spare1.selectJobStatus[7].completed,
             hmiInterface := "Unit1.Em2.HmiInterface".semiAutoSplice.jobs,
             jobs := "Unit1.Em2.ControlNodes".semiAutoSplice.jobs,
             jobStatus => "Unit1.EmNodes".emRelations.em02.sequence.Spare1.selectJobStatus[8]);
END_REGION

REGION Network 24: Select Job [9]
   RUNG wire#powerrail
      #instJob9(interlock := wire#w1, startCondition := wire#w2, parentReferenceDesignator := "Unit1.Em2.Config".em.referenceDesignator.combined, jobNumber := "U1EM2_JOB09", singleCycleJob := TRUE, hmiInterface := "Unit1.Em2.HmiInterface".semiAutoSplice.jobs, jobs := "Unit1.Em2.ControlNodes".semiAutoSplice.jobs, jobStatus => "Unit1.EmNodes".emRelations.em02.sequence.Spare1.selectJobStatus[9])
   END_RUNG
   RUNG wire#powerrail
      I_Contact( "Unit1.Em2.Alarms".emAlarms.error )
   END_RUNG wire#w1
   RUNG wire#powerrail
      Contact( #statUnitStatus.mode.production )
      Contact( #statUnitStatus.state.execute )
      Contact( "Unit1.EmNodes".emRelations.em02.sequence.Spare1.selectJobStatus[8].completed )
      Contact( #FALSE )
   END_RUNG wire#w2
   // the same network as SCL:
   #instJob9(parentReferenceDesignator := "Unit1.Em2.Config".em.referenceDesignator.combined,   // "LAF_SelectJob"
             jobNumber := "U1EM2_JOB09",
             singleCycleJob := TRUE,
             interlock := NOT "Unit1.Em2.Alarms".emAlarms.error,
             startCondition := #statUnitStatus.mode.production AND #statUnitStatus.state.execute AND "Unit1.EmNodes".emRelations.em02.sequence.Spare1.selectJobStatus[8].completed AND #FALSE,
             hmiInterface := "Unit1.Em2.HmiInterface".semiAutoSplice.jobs,
             jobs := "Unit1.Em2.ControlNodes".semiAutoSplice.jobs,
             jobStatus => "Unit1.EmNodes".emRelations.em02.sequence.Spare1.selectJobStatus[9]);
END_REGION

REGION Network 25: Select Job [10] Top to Btm : TOP Vacc Off & Btm Vacc On
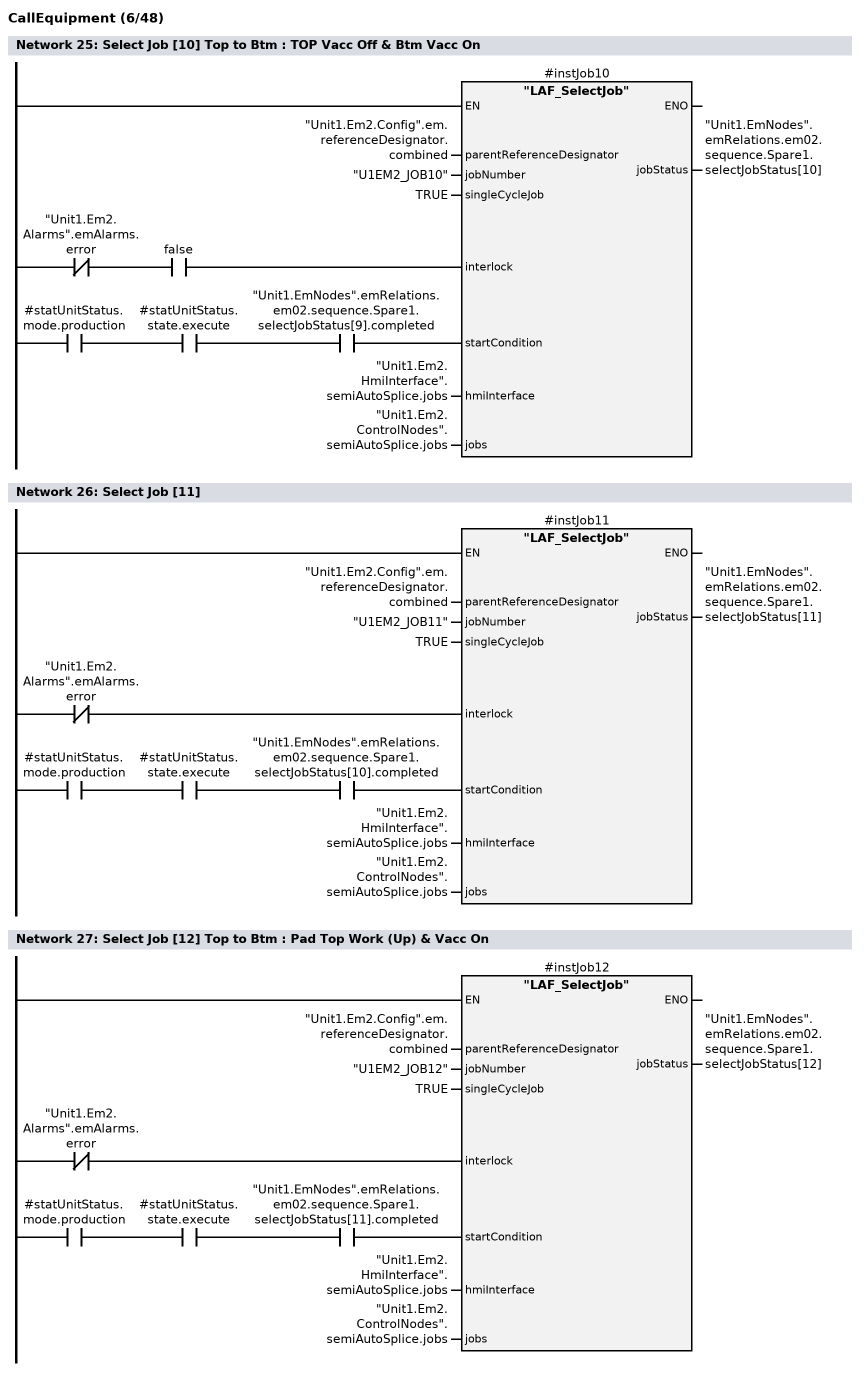
   RUNG wire#powerrail
      #instJob10(interlock := wire#w1, startCondition := wire#w2, parentReferenceDesignator := "Unit1.Em2.Config".em.referenceDesignator.combined, jobNumber := "U1EM2_JOB10", singleCycleJob := TRUE, hmiInterface := "Unit1.Em2.HmiInterface".semiAutoSplice.jobs, jobs := "Unit1.Em2.ControlNodes".semiAutoSplice.jobs, jobStatus => "Unit1.EmNodes".emRelations.em02.sequence.Spare1.selectJobStatus[10])
   END_RUNG
   RUNG wire#powerrail
      I_Contact( "Unit1.Em2.Alarms".emAlarms.error )
      Contact( false )
   END_RUNG wire#w1
   RUNG wire#powerrail
      Contact( #statUnitStatus.mode.production )
      Contact( #statUnitStatus.state.execute )
      Contact( "Unit1.EmNodes".emRelations.em02.sequence.Spare1.selectJobStatus[9].completed )
   END_RUNG wire#w2
   // the same network as SCL:
   #instJob10(parentReferenceDesignator := "Unit1.Em2.Config".em.referenceDesignator.combined,   // "LAF_SelectJob"
              jobNumber := "U1EM2_JOB10",
              singleCycleJob := TRUE,
              interlock := NOT "Unit1.Em2.Alarms".emAlarms.error AND false,
              startCondition := #statUnitStatus.mode.production AND #statUnitStatus.state.execute AND "Unit1.EmNodes".emRelations.em02.sequence.Spare1.selectJobStatus[9].completed,
              hmiInterface := "Unit1.Em2.HmiInterface".semiAutoSplice.jobs,
              jobs := "Unit1.Em2.ControlNodes".semiAutoSplice.jobs,
              jobStatus => "Unit1.EmNodes".emRelations.em02.sequence.Spare1.selectJobStatus[10]);
END_REGION

REGION Network 26: Select Job [11]
   RUNG wire#powerrail
      #instJob11(interlock := wire#w1, startCondition := wire#w2, parentReferenceDesignator := "Unit1.Em2.Config".em.referenceDesignator.combined, jobNumber := "U1EM2_JOB11", singleCycleJob := TRUE, hmiInterface := "Unit1.Em2.HmiInterface".semiAutoSplice.jobs, jobs := "Unit1.Em2.ControlNodes".semiAutoSplice.jobs, jobStatus => "Unit1.EmNodes".emRelations.em02.sequence.Spare1.selectJobStatus[11])
   END_RUNG
   RUNG wire#powerrail
      I_Contact( "Unit1.Em2.Alarms".emAlarms.error )
   END_RUNG wire#w1
   RUNG wire#powerrail
      Contact( #statUnitStatus.mode.production )
      Contact( #statUnitStatus.state.execute )
      Contact( "Unit1.EmNodes".emRelations.em02.sequence.Spare1.selectJobStatus[10].completed )
   END_RUNG wire#w2
   // the same network as SCL:
   #instJob11(parentReferenceDesignator := "Unit1.Em2.Config".em.referenceDesignator.combined,   // "LAF_SelectJob"
              jobNumber := "U1EM2_JOB11",
              singleCycleJob := TRUE,
              interlock := NOT "Unit1.Em2.Alarms".emAlarms.error,
              startCondition := #statUnitStatus.mode.production AND #statUnitStatus.state.execute AND "Unit1.EmNodes".emRelations.em02.sequence.Spare1.selectJobStatus[10].completed,
              hmiInterface := "Unit1.Em2.HmiInterface".semiAutoSplice.jobs,
              jobs := "Unit1.Em2.ControlNodes".semiAutoSplice.jobs,
              jobStatus => "Unit1.EmNodes".emRelations.em02.sequence.Spare1.selectJobStatus[11]);
END_REGION

REGION Network 27: Select Job [12] Top to Btm : Pad Top Work (Up) & Vacc On
   RUNG wire#powerrail
      #instJob12(interlock := wire#w1, startCondition := wire#w2, parentReferenceDesignator := "Unit1.Em2.Config".em.referenceDesignator.combined, jobNumber := "U1EM2_JOB12", singleCycleJob := TRUE, hmiInterface := "Unit1.Em2.HmiInterface".semiAutoSplice.jobs, jobs := "Unit1.Em2.ControlNodes".semiAutoSplice.jobs, jobStatus => "Unit1.EmNodes".emRelations.em02.sequence.Spare1.selectJobStatus[12])
   END_RUNG
   RUNG wire#powerrail
      I_Contact( "Unit1.Em2.Alarms".emAlarms.error )
   END_RUNG wire#w1
   RUNG wire#powerrail
      Contact( #statUnitStatus.mode.production )
      Contact( #statUnitStatus.state.execute )
      Contact( "Unit1.EmNodes".emRelations.em02.sequence.Spare1.selectJobStatus[11].completed )
   END_RUNG wire#w2
   // the same network as SCL:
   #instJob12(parentReferenceDesignator := "Unit1.Em2.Config".em.referenceDesignator.combined,   // "LAF_SelectJob"
              jobNumber := "U1EM2_JOB12",
              singleCycleJob := TRUE,
              interlock := NOT "Unit1.Em2.Alarms".emAlarms.error,
              startCondition := #statUnitStatus.mode.production AND #statUnitStatus.state.execute AND "Unit1.EmNodes".emRelations.em02.sequence.Spare1.selectJobStatus[11].completed,
              hmiInterface := "Unit1.Em2.HmiInterface".semiAutoSplice.jobs,
              jobs := "Unit1.Em2.ControlNodes".semiAutoSplice.jobs,
              jobStatus => "Unit1.EmNodes".emRelations.em02.sequence.Spare1.selectJobStatus[12]);
END_REGION

REGION Network 28: Select Job [13] Top to Btm : BTM Vacc Off & Pad Btm Home (Down)
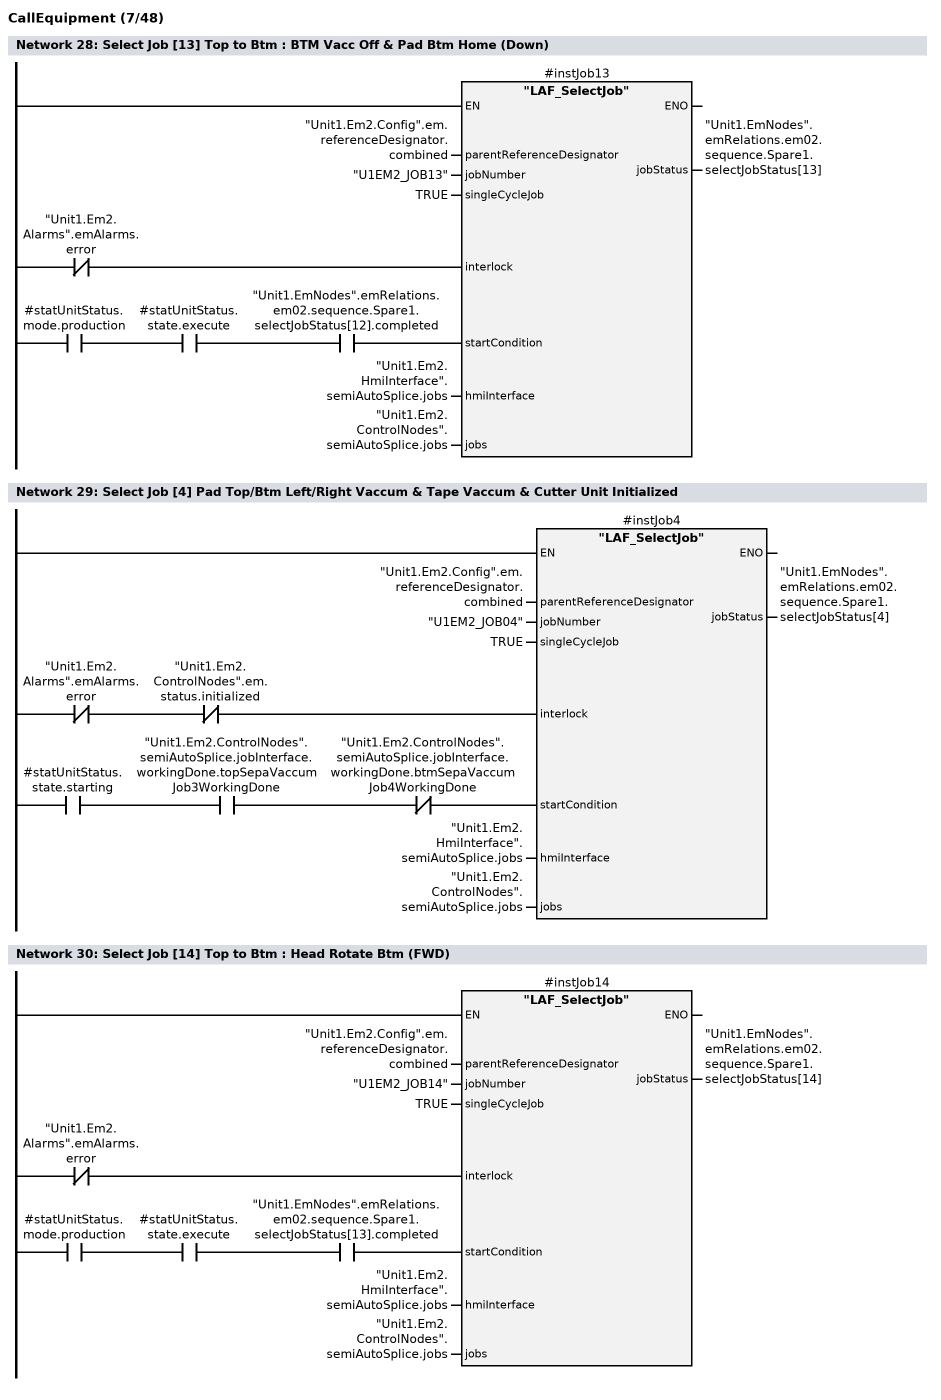
   RUNG wire#powerrail
      #instJob13(interlock := wire#w1, startCondition := wire#w2, parentReferenceDesignator := "Unit1.Em2.Config".em.referenceDesignator.combined, jobNumber := "U1EM2_JOB13", singleCycleJob := TRUE, hmiInterface := "Unit1.Em2.HmiInterface".semiAutoSplice.jobs, jobs := "Unit1.Em2.ControlNodes".semiAutoSplice.jobs, jobStatus => "Unit1.EmNodes".emRelations.em02.sequence.Spare1.selectJobStatus[13])
   END_RUNG
   RUNG wire#powerrail
      I_Contact( "Unit1.Em2.Alarms".emAlarms.error )
   END_RUNG wire#w1
   RUNG wire#powerrail
      Contact( #statUnitStatus.mode.production )
      Contact( #statUnitStatus.state.execute )
      Contact( "Unit1.EmNodes".emRelations.em02.sequence.Spare1.selectJobStatus[12].completed )
   END_RUNG wire#w2
   // the same network as SCL:
   #instJob13(parentReferenceDesignator := "Unit1.Em2.Config".em.referenceDesignator.combined,   // "LAF_SelectJob"
              jobNumber := "U1EM2_JOB13",
              singleCycleJob := TRUE,
              interlock := NOT "Unit1.Em2.Alarms".emAlarms.error,
              startCondition := #statUnitStatus.mode.production AND #statUnitStatus.state.execute AND "Unit1.EmNodes".emRelations.em02.sequence.Spare1.selectJobStatus[12].completed,
              hmiInterface := "Unit1.Em2.HmiInterface".semiAutoSplice.jobs,
              jobs := "Unit1.Em2.ControlNodes".semiAutoSplice.jobs,
              jobStatus => "Unit1.EmNodes".emRelations.em02.sequence.Spare1.selectJobStatus[13]);
END_REGION

REGION Network 29: Select Job [4] Pad Top/Btm Left/Right Vaccum & Tape Vaccum & Cutter Unit Initialized
   RUNG wire#powerrail
      #instJob4(interlock := wire#w1, startCondition := wire#w2, parentReferenceDesignator := "Unit1.Em2.Config".em.referenceDesignator.combined, jobNumber := "U1EM2_JOB04", singleCycleJob := TRUE, hmiInterface := "Unit1.Em2.HmiInterface".semiAutoSplice.jobs, jobs := "Unit1.Em2.ControlNodes".semiAutoSplice.jobs, jobStatus => "Unit1.EmNodes".emRelations.em02.sequence.Spare1.selectJobStatus[4])
   END_RUNG
   RUNG wire#powerrail
      I_Contact( "Unit1.Em2.Alarms".emAlarms.error )
      I_Contact( "Unit1.Em2.ControlNodes".em.status.initialized )
   END_RUNG wire#w1
   RUNG wire#powerrail
      Contact( #statUnitStatus.state.starting )
      Contact( "Unit1.Em2.ControlNodes".semiAutoSplice.jobInterface.workingDone.topSepaVaccumJob3WorkingDone )
      I_Contact( "Unit1.Em2.ControlNodes".semiAutoSplice.jobInterface.workingDone.btmSepaVaccumJob4WorkingDone )
   END_RUNG wire#w2
   // the same network as SCL:
   #instJob4(parentReferenceDesignator := "Unit1.Em2.Config".em.referenceDesignator.combined,   // "LAF_SelectJob"
             jobNumber := "U1EM2_JOB04",
             singleCycleJob := TRUE,
             interlock := NOT "Unit1.Em2.Alarms".emAlarms.error AND NOT "Unit1.Em2.ControlNodes".em.status.initialized,
             startCondition := #statUnitStatus.state.starting AND "Unit1.Em2.ControlNodes".semiAutoSplice.jobInterface.workingDone.topSepaVaccumJob3WorkingDone AND NOT "Unit1.Em2.ControlNodes".semiAutoSplice.jobInterface.workingDone.btmSepaVaccumJob4WorkingDone,
             hmiInterface := "Unit1.Em2.HmiInterface".semiAutoSplice.jobs,
             jobs := "Unit1.Em2.ControlNodes".semiAutoSplice.jobs,
             jobStatus => "Unit1.EmNodes".emRelations.em02.sequence.Spare1.selectJobStatus[4]);
END_REGION

REGION Network 30: Select Job [14] Top to Btm : Head Rotate Btm (FWD)
   RUNG wire#powerrail
      #instJob14(interlock := wire#w1, startCondition := wire#w2, parentReferenceDesignator := "Unit1.Em2.Config".em.referenceDesignator.combined, jobNumber := "U1EM2_JOB14", singleCycleJob := TRUE, hmiInterface := "Unit1.Em2.HmiInterface".semiAutoSplice.jobs, jobs := "Unit1.Em2.ControlNodes".semiAutoSplice.jobs, jobStatus => "Unit1.EmNodes".emRelations.em02.sequence.Spare1.selectJobStatus[14])
   END_RUNG
   RUNG wire#powerrail
      I_Contact( "Unit1.Em2.Alarms".emAlarms.error )
   END_RUNG wire#w1
   RUNG wire#powerrail
      Contact( #statUnitStatus.mode.production )
      Contact( #statUnitStatus.state.execute )
      Contact( "Unit1.EmNodes".emRelations.em02.sequence.Spare1.selectJobStatus[13].completed )
   END_RUNG wire#w2
   // the same network as SCL:
   #instJob14(parentReferenceDesignator := "Unit1.Em2.Config".em.referenceDesignator.combined,   // "LAF_SelectJob"
              jobNumber := "U1EM2_JOB14",
              singleCycleJob := TRUE,
              interlock := NOT "Unit1.Em2.Alarms".emAlarms.error,
              startCondition := #statUnitStatus.mode.production AND #statUnitStatus.state.execute AND "Unit1.EmNodes".emRelations.em02.sequence.Spare1.selectJobStatus[13].completed,
              hmiInterface := "Unit1.Em2.HmiInterface".semiAutoSplice.jobs,
              jobs := "Unit1.Em2.ControlNodes".semiAutoSplice.jobs,
              jobStatus => "Unit1.EmNodes".emRelations.em02.sequence.Spare1.selectJobStatus[14]);
END_REGION

REGION Network 31: Select Job [15] Top to Btm : TAPPING
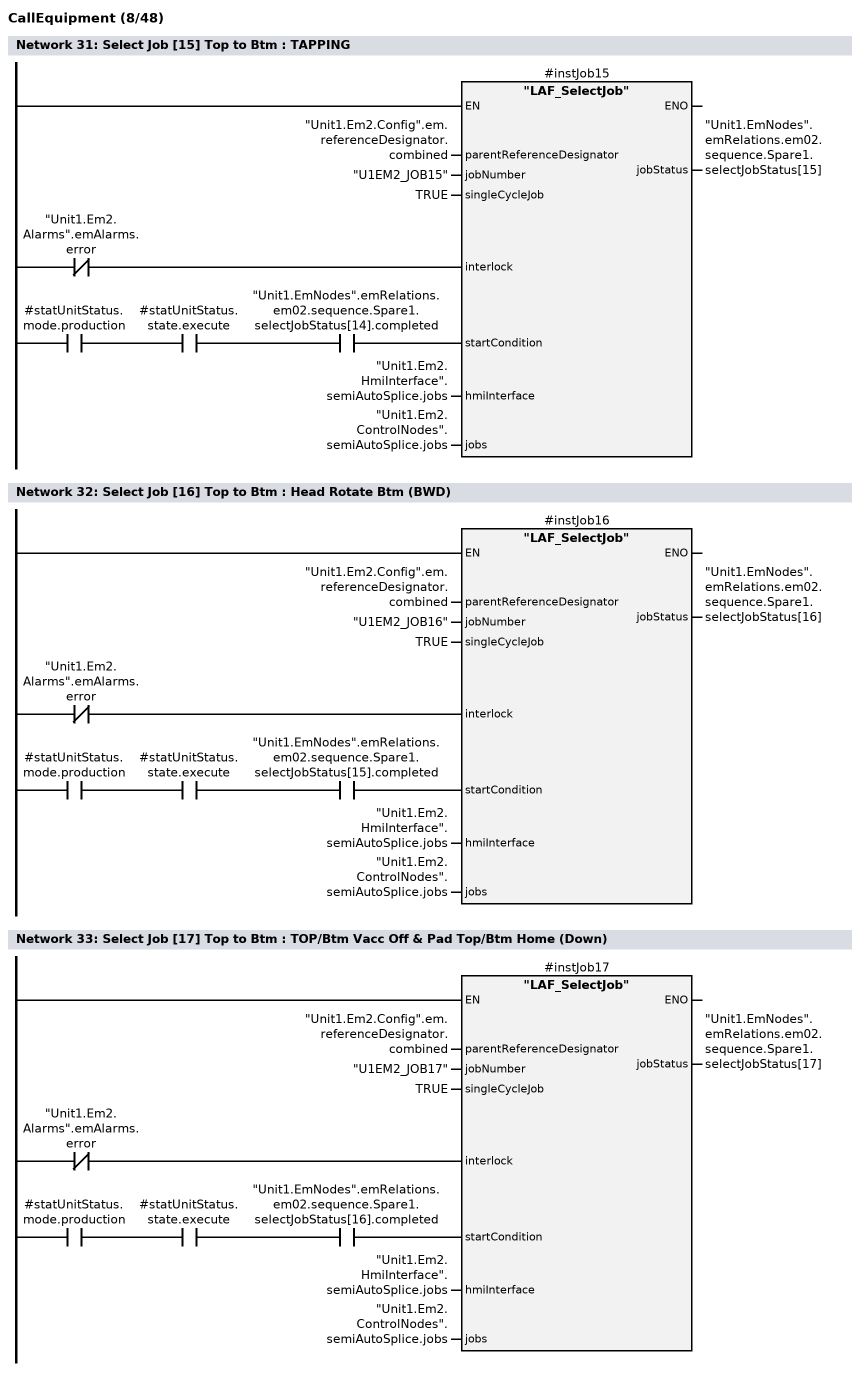
   RUNG wire#powerrail
      #instJob15(interlock := wire#w1, startCondition := wire#w2, parentReferenceDesignator := "Unit1.Em2.Config".em.referenceDesignator.combined, jobNumber := "U1EM2_JOB15", singleCycleJob := TRUE, hmiInterface := "Unit1.Em2.HmiInterface".semiAutoSplice.jobs, jobs := "Unit1.Em2.ControlNodes".semiAutoSplice.jobs, jobStatus => "Unit1.EmNodes".emRelations.em02.sequence.Spare1.selectJobStatus[15])
   END_RUNG
   RUNG wire#powerrail
      I_Contact( "Unit1.Em2.Alarms".emAlarms.error )
   END_RUNG wire#w1
   RUNG wire#powerrail
      Contact( #statUnitStatus.mode.production )
      Contact( #statUnitStatus.state.execute )
      Contact( "Unit1.EmNodes".emRelations.em02.sequence.Spare1.selectJobStatus[14].completed )
   END_RUNG wire#w2
   // the same network as SCL:
   #instJob15(parentReferenceDesignator := "Unit1.Em2.Config".em.referenceDesignator.combined,   // "LAF_SelectJob"
              jobNumber := "U1EM2_JOB15",
              singleCycleJob := TRUE,
              interlock := NOT "Unit1.Em2.Alarms".emAlarms.error,
              startCondition := #statUnitStatus.mode.production AND #statUnitStatus.state.execute AND "Unit1.EmNodes".emRelations.em02.sequence.Spare1.selectJobStatus[14].completed,
              hmiInterface := "Unit1.Em2.HmiInterface".semiAutoSplice.jobs,
              jobs := "Unit1.Em2.ControlNodes".semiAutoSplice.jobs,
              jobStatus => "Unit1.EmNodes".emRelations.em02.sequence.Spare1.selectJobStatus[15]);
END_REGION

REGION Network 32: Select Job [16] Top to Btm : Head Rotate Btm (BWD)
   RUNG wire#powerrail
      #instJob16(interlock := wire#w1, startCondition := wire#w2, parentReferenceDesignator := "Unit1.Em2.Config".em.referenceDesignator.combined, jobNumber := "U1EM2_JOB16", singleCycleJob := TRUE, hmiInterface := "Unit1.Em2.HmiInterface".semiAutoSplice.jobs, jobs := "Unit1.Em2.ControlNodes".semiAutoSplice.jobs, jobStatus => "Unit1.EmNodes".emRelations.em02.sequence.Spare1.selectJobStatus[16])
   END_RUNG
   RUNG wire#powerrail
      I_Contact( "Unit1.Em2.Alarms".emAlarms.error )
   END_RUNG wire#w1
   RUNG wire#powerrail
      Contact( #statUnitStatus.mode.production )
      Contact( #statUnitStatus.state.execute )
      Contact( "Unit1.EmNodes".emRelations.em02.sequence.Spare1.selectJobStatus[15].completed )
   END_RUNG wire#w2
   // the same network as SCL:
   #instJob16(parentReferenceDesignator := "Unit1.Em2.Config".em.referenceDesignator.combined,   // "LAF_SelectJob"
              jobNumber := "U1EM2_JOB16",
              singleCycleJob := TRUE,
              interlock := NOT "Unit1.Em2.Alarms".emAlarms.error,
              startCondition := #statUnitStatus.mode.production AND #statUnitStatus.state.execute AND "Unit1.EmNodes".emRelations.em02.sequence.Spare1.selectJobStatus[15].completed,
              hmiInterface := "Unit1.Em2.HmiInterface".semiAutoSplice.jobs,
              jobs := "Unit1.Em2.ControlNodes".semiAutoSplice.jobs,
              jobStatus => "Unit1.EmNodes".emRelations.em02.sequence.Spare1.selectJobStatus[16]);
END_REGION

REGION Network 33: Select Job [17] Top to Btm : TOP/Btm Vacc Off & Pad Top/Btm Home (Down)
   RUNG wire#powerrail
      #instJob17(interlock := wire#w1, startCondition := wire#w2, parentReferenceDesignator := "Unit1.Em2.Config".em.referenceDesignator.combined, jobNumber := "U1EM2_JOB17", singleCycleJob := TRUE, hmiInterface := "Unit1.Em2.HmiInterface".semiAutoSplice.jobs, jobs := "Unit1.Em2.ControlNodes".semiAutoSplice.jobs, jobStatus => "Unit1.EmNodes".emRelations.em02.sequence.Spare1.selectJobStatus[17])
   END_RUNG
   RUNG wire#powerrail
      I_Contact( "Unit1.Em2.Alarms".emAlarms.error )
   END_RUNG wire#w1
   RUNG wire#powerrail
      Contact( #statUnitStatus.mode.production )
      Contact( #statUnitStatus.state.execute )
      Contact( "Unit1.EmNodes".emRelations.em02.sequence.Spare1.selectJobStatus[16].completed )
   END_RUNG wire#w2
   // the same network as SCL:
   #instJob17(parentReferenceDesignator := "Unit1.Em2.Config".em.referenceDesignator.combined,   // "LAF_SelectJob"
              jobNumber := "U1EM2_JOB17",
              singleCycleJob := TRUE,
              interlock := NOT "Unit1.Em2.Alarms".emAlarms.error,
              startCondition := #statUnitStatus.mode.production AND #statUnitStatus.state.execute AND "Unit1.EmNodes".emRelations.em02.sequence.Spare1.selectJobStatus[16].completed,
              hmiInterface := "Unit1.Em2.HmiInterface".semiAutoSplice.jobs,
              jobs := "Unit1.Em2.ControlNodes".semiAutoSplice.jobs,
              jobStatus => "Unit1.EmNodes".emRelations.em02.sequence.Spare1.selectJobStatus[17]);
END_REGION

REGION Network 34: Select Job [18] Top to Btm : Link Change
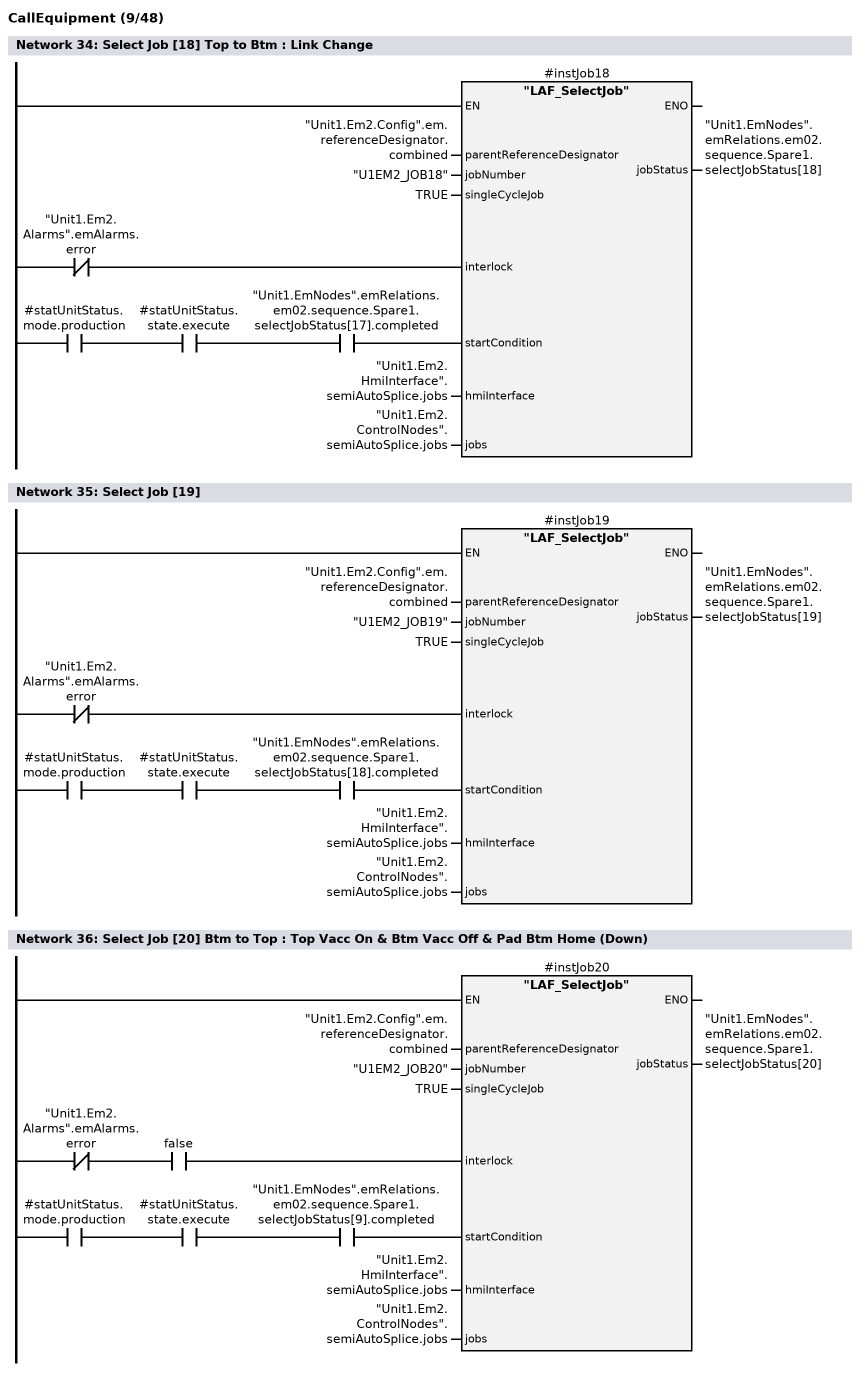
   RUNG wire#powerrail
      #instJob18(interlock := wire#w1, startCondition := wire#w2, parentReferenceDesignator := "Unit1.Em2.Config".em.referenceDesignator.combined, jobNumber := "U1EM2_JOB18", singleCycleJob := TRUE, hmiInterface := "Unit1.Em2.HmiInterface".semiAutoSplice.jobs, jobs := "Unit1.Em2.ControlNodes".semiAutoSplice.jobs, jobStatus => "Unit1.EmNodes".emRelations.em02.sequence.Spare1.selectJobStatus[18])
   END_RUNG
   RUNG wire#powerrail
      I_Contact( "Unit1.Em2.Alarms".emAlarms.error )
   END_RUNG wire#w1
   RUNG wire#powerrail
      Contact( #statUnitStatus.mode.production )
      Contact( #statUnitStatus.state.execute )
      Contact( "Unit1.EmNodes".emRelations.em02.sequence.Spare1.selectJobStatus[17].completed )
   END_RUNG wire#w2
   // the same network as SCL:
   #instJob18(parentReferenceDesignator := "Unit1.Em2.Config".em.referenceDesignator.combined,   // "LAF_SelectJob"
              jobNumber := "U1EM2_JOB18",
              singleCycleJob := TRUE,
              interlock := NOT "Unit1.Em2.Alarms".emAlarms.error,
              startCondition := #statUnitStatus.mode.production AND #statUnitStatus.state.execute AND "Unit1.EmNodes".emRelations.em02.sequence.Spare1.selectJobStatus[17].completed,
              hmiInterface := "Unit1.Em2.HmiInterface".semiAutoSplice.jobs,
              jobs := "Unit1.Em2.ControlNodes".semiAutoSplice.jobs,
              jobStatus => "Unit1.EmNodes".emRelations.em02.sequence.Spare1.selectJobStatus[18]);
END_REGION

REGION Network 35: Select Job [19]
   RUNG wire#powerrail
      #instJob19(interlock := wire#w1, startCondition := wire#w2, parentReferenceDesignator := "Unit1.Em2.Config".em.referenceDesignator.combined, jobNumber := "U1EM2_JOB19", singleCycleJob := TRUE, hmiInterface := "Unit1.Em2.HmiInterface".semiAutoSplice.jobs, jobs := "Unit1.Em2.ControlNodes".semiAutoSplice.jobs, jobStatus => "Unit1.EmNodes".emRelations.em02.sequence.Spare1.selectJobStatus[19])
   END_RUNG
   RUNG wire#powerrail
      I_Contact( "Unit1.Em2.Alarms".emAlarms.error )
   END_RUNG wire#w1
   RUNG wire#powerrail
      Contact( #statUnitStatus.mode.production )
      Contact( #statUnitStatus.state.execute )
      Contact( "Unit1.EmNodes".emRelations.em02.sequence.Spare1.selectJobStatus[18].completed )
   END_RUNG wire#w2
   // the same network as SCL:
   #instJob19(parentReferenceDesignator := "Unit1.Em2.Config".em.referenceDesignator.combined,   // "LAF_SelectJob"
              jobNumber := "U1EM2_JOB19",
              singleCycleJob := TRUE,
              interlock := NOT "Unit1.Em2.Alarms".emAlarms.error,
              startCondition := #statUnitStatus.mode.production AND #statUnitStatus.state.execute AND "Unit1.EmNodes".emRelations.em02.sequence.Spare1.selectJobStatus[18].completed,
              hmiInterface := "Unit1.Em2.HmiInterface".semiAutoSplice.jobs,
              jobs := "Unit1.Em2.ControlNodes".semiAutoSplice.jobs,
              jobStatus => "Unit1.EmNodes".emRelations.em02.sequence.Spare1.selectJobStatus[19]);
END_REGION

REGION Network 36: Select Job [20] Btm to Top : Top Vacc On & Btm Vacc Off & Pad Btm Home (Down)
   RUNG wire#powerrail
      #instJob20(interlock := wire#w1, startCondition := wire#w2, parentReferenceDesignator := "Unit1.Em2.Config".em.referenceDesignator.combined, jobNumber := "U1EM2_JOB20", singleCycleJob := TRUE, hmiInterface := "Unit1.Em2.HmiInterface".semiAutoSplice.jobs, jobs := "Unit1.Em2.ControlNodes".semiAutoSplice.jobs, jobStatus => "Unit1.EmNodes".emRelations.em02.sequence.Spare1.selectJobStatus[20])
   END_RUNG
   RUNG wire#powerrail
      I_Contact( "Unit1.Em2.Alarms".emAlarms.error )
      Contact( false )
   END_RUNG wire#w1
   RUNG wire#powerrail
      Contact( #statUnitStatus.mode.production )
      Contact( #statUnitStatus.state.execute )
      Contact( "Unit1.EmNodes".emRelations.em02.sequence.Spare1.selectJobStatus[9].completed )
   END_RUNG wire#w2
   // the same network as SCL:
   #instJob20(parentReferenceDesignator := "Unit1.Em2.Config".em.referenceDesignator.combined,   // "LAF_SelectJob"
              jobNumber := "U1EM2_JOB20",
              singleCycleJob := TRUE,
              interlock := NOT "Unit1.Em2.Alarms".emAlarms.error AND false,
              startCondition := #statUnitStatus.mode.production AND #statUnitStatus.state.execute AND "Unit1.EmNodes".emRelations.em02.sequence.Spare1.selectJobStatus[9].completed,
              hmiInterface := "Unit1.Em2.HmiInterface".semiAutoSplice.jobs,
              jobs := "Unit1.Em2.ControlNodes".semiAutoSplice.jobs,
              jobStatus => "Unit1.EmNodes".emRelations.em02.sequence.Spare1.selectJobStatus[20]);
END_REGION

REGION Network 37: Select Job [21]
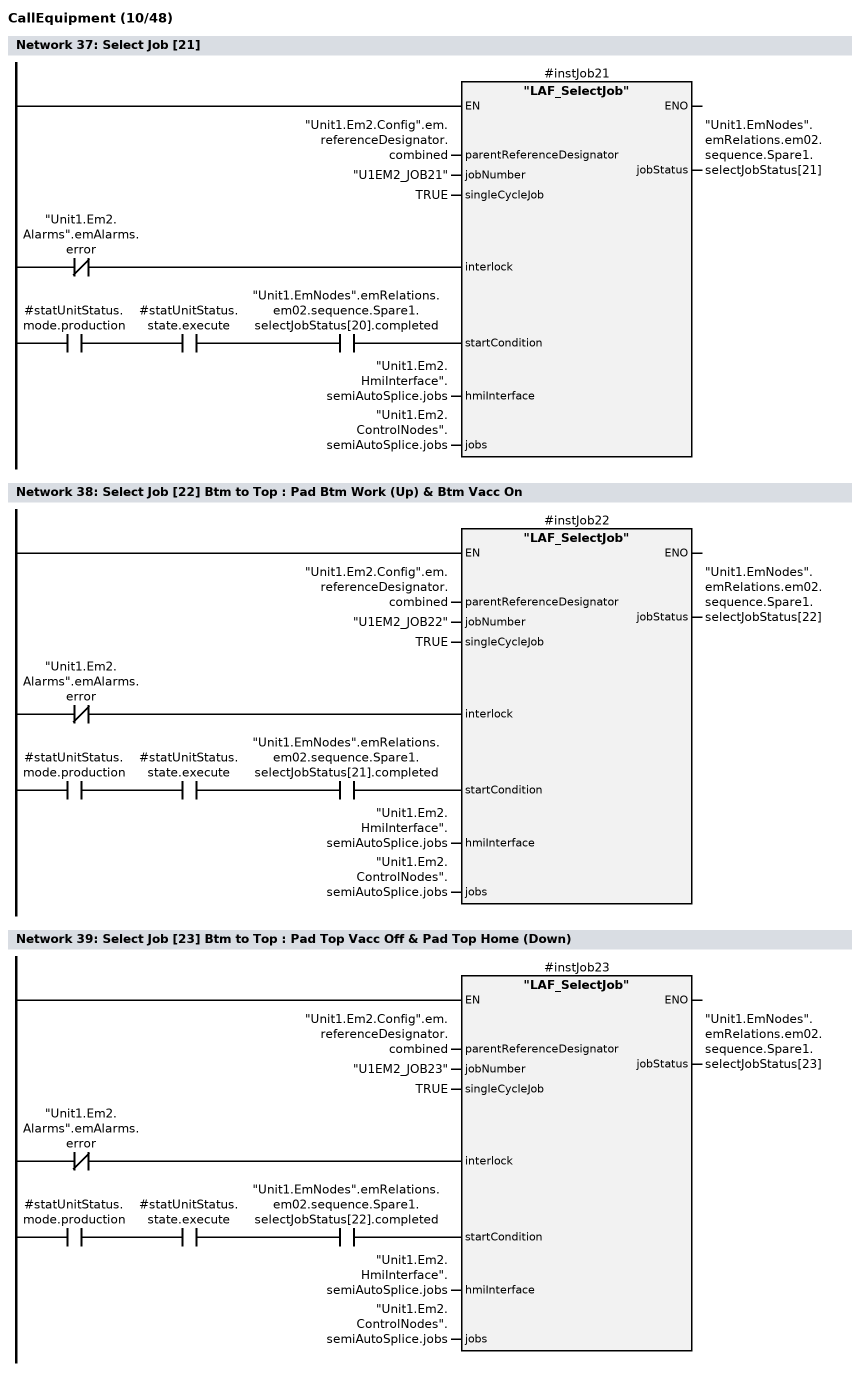
   RUNG wire#powerrail
      #instJob21(interlock := wire#w1, startCondition := wire#w2, parentReferenceDesignator := "Unit1.Em2.Config".em.referenceDesignator.combined, jobNumber := "U1EM2_JOB21", singleCycleJob := TRUE, hmiInterface := "Unit1.Em2.HmiInterface".semiAutoSplice.jobs, jobs := "Unit1.Em2.ControlNodes".semiAutoSplice.jobs, jobStatus => "Unit1.EmNodes".emRelations.em02.sequence.Spare1.selectJobStatus[21])
   END_RUNG
   RUNG wire#powerrail
      I_Contact( "Unit1.Em2.Alarms".emAlarms.error )
   END_RUNG wire#w1
   RUNG wire#powerrail
      Contact( #statUnitStatus.mode.production )
      Contact( #statUnitStatus.state.execute )
      Contact( "Unit1.EmNodes".emRelations.em02.sequence.Spare1.selectJobStatus[20].completed )
   END_RUNG wire#w2
   // the same network as SCL:
   #instJob21(parentReferenceDesignator := "Unit1.Em2.Config".em.referenceDesignator.combined,   // "LAF_SelectJob"
              jobNumber := "U1EM2_JOB21",
              singleCycleJob := TRUE,
              interlock := NOT "Unit1.Em2.Alarms".emAlarms.error,
              startCondition := #statUnitStatus.mode.production AND #statUnitStatus.state.execute AND "Unit1.EmNodes".emRelations.em02.sequence.Spare1.selectJobStatus[20].completed,
              hmiInterface := "Unit1.Em2.HmiInterface".semiAutoSplice.jobs,
              jobs := "Unit1.Em2.ControlNodes".semiAutoSplice.jobs,
              jobStatus => "Unit1.EmNodes".emRelations.em02.sequence.Spare1.selectJobStatus[21]);
END_REGION

REGION Network 38: Select Job [22] Btm to Top : Pad Btm Work (Up) & Btm Vacc On
   RUNG wire#powerrail
      #instJob22(interlock := wire#w1, startCondition := wire#w2, parentReferenceDesignator := "Unit1.Em2.Config".em.referenceDesignator.combined, jobNumber := "U1EM2_JOB22", singleCycleJob := TRUE, hmiInterface := "Unit1.Em2.HmiInterface".semiAutoSplice.jobs, jobs := "Unit1.Em2.ControlNodes".semiAutoSplice.jobs, jobStatus => "Unit1.EmNodes".emRelations.em02.sequence.Spare1.selectJobStatus[22])
   END_RUNG
   RUNG wire#powerrail
      I_Contact( "Unit1.Em2.Alarms".emAlarms.error )
   END_RUNG wire#w1
   RUNG wire#powerrail
      Contact( #statUnitStatus.mode.production )
      Contact( #statUnitStatus.state.execute )
      Contact( "Unit1.EmNodes".emRelations.em02.sequence.Spare1.selectJobStatus[21].completed )
   END_RUNG wire#w2
   // the same network as SCL:
   #instJob22(parentReferenceDesignator := "Unit1.Em2.Config".em.referenceDesignator.combined,   // "LAF_SelectJob"
              jobNumber := "U1EM2_JOB22",
              singleCycleJob := TRUE,
              interlock := NOT "Unit1.Em2.Alarms".emAlarms.error,
              startCondition := #statUnitStatus.mode.production AND #statUnitStatus.state.execute AND "Unit1.EmNodes".emRelations.em02.sequence.Spare1.selectJobStatus[21].completed,
              hmiInterface := "Unit1.Em2.HmiInterface".semiAutoSplice.jobs,
              jobs := "Unit1.Em2.ControlNodes".semiAutoSplice.jobs,
              jobStatus => "Unit1.EmNodes".emRelations.em02.sequence.Spare1.selectJobStatus[22]);
END_REGION

REGION Network 39: Select Job [23] Btm to Top : Pad Top Vacc Off & Pad Top Home (Down)
   RUNG wire#powerrail
      #instJob23(interlock := wire#w1, startCondition := wire#w2, parentReferenceDesignator := "Unit1.Em2.Config".em.referenceDesignator.combined, jobNumber := "U1EM2_JOB23", singleCycleJob := TRUE, hmiInterface := "Unit1.Em2.HmiInterface".semiAutoSplice.jobs, jobs := "Unit1.Em2.ControlNodes".semiAutoSplice.jobs, jobStatus => "Unit1.EmNodes".emRelations.em02.sequence.Spare1.selectJobStatus[23])
   END_RUNG
   RUNG wire#powerrail
      I_Contact( "Unit1.Em2.Alarms".emAlarms.error )
   END_RUNG wire#w1
   RUNG wire#powerrail
      Contact( #statUnitStatus.mode.production )
      Contact( #statUnitStatus.state.execute )
      Contact( "Unit1.EmNodes".emRelations.em02.sequence.Spare1.selectJobStatus[22].completed )
   END_RUNG wire#w2
   // the same network as SCL:
   #instJob23(parentReferenceDesignator := "Unit1.Em2.Config".em.referenceDesignator.combined,   // "LAF_SelectJob"
              jobNumber := "U1EM2_JOB23",
              singleCycleJob := TRUE,
              interlock := NOT "Unit1.Em2.Alarms".emAlarms.error,
              startCondition := #statUnitStatus.mode.production AND #statUnitStatus.state.execute AND "Unit1.EmNodes".emRelations.em02.sequence.Spare1.selectJobStatus[22].completed,
              hmiInterface := "Unit1.Em2.HmiInterface".semiAutoSplice.jobs,
              jobs := "Unit1.Em2.ControlNodes".semiAutoSplice.jobs,
              jobStatus => "Unit1.EmNodes".emRelations.em02.sequence.Spare1.selectJobStatus[23]);
END_REGION

REGION Network 40: Select Job [24] Btm to Top : Head Rotate Top (FWD)
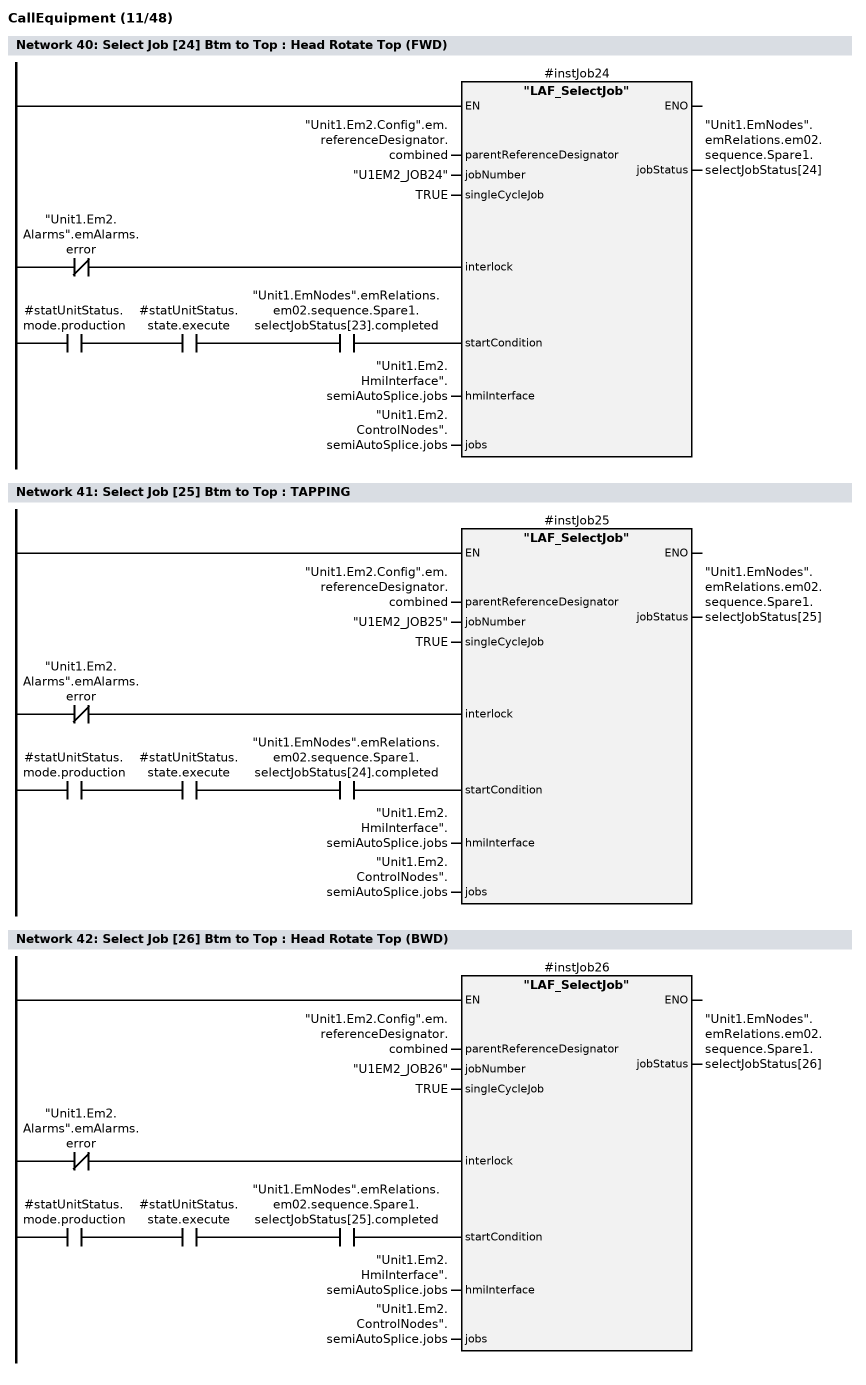
   RUNG wire#powerrail
      #instJob24(interlock := wire#w1, startCondition := wire#w2, parentReferenceDesignator := "Unit1.Em2.Config".em.referenceDesignator.combined, jobNumber := "U1EM2_JOB24", singleCycleJob := TRUE, hmiInterface := "Unit1.Em2.HmiInterface".semiAutoSplice.jobs, jobs := "Unit1.Em2.ControlNodes".semiAutoSplice.jobs, jobStatus => "Unit1.EmNodes".emRelations.em02.sequence.Spare1.selectJobStatus[24])
   END_RUNG
   RUNG wire#powerrail
      I_Contact( "Unit1.Em2.Alarms".emAlarms.error )
   END_RUNG wire#w1
   RUNG wire#powerrail
      Contact( #statUnitStatus.mode.production )
      Contact( #statUnitStatus.state.execute )
      Contact( "Unit1.EmNodes".emRelations.em02.sequence.Spare1.selectJobStatus[23].completed )
   END_RUNG wire#w2
   // the same network as SCL:
   #instJob24(parentReferenceDesignator := "Unit1.Em2.Config".em.referenceDesignator.combined,   // "LAF_SelectJob"
              jobNumber := "U1EM2_JOB24",
              singleCycleJob := TRUE,
              interlock := NOT "Unit1.Em2.Alarms".emAlarms.error,
              startCondition := #statUnitStatus.mode.production AND #statUnitStatus.state.execute AND "Unit1.EmNodes".emRelations.em02.sequence.Spare1.selectJobStatus[23].completed,
              hmiInterface := "Unit1.Em2.HmiInterface".semiAutoSplice.jobs,
              jobs := "Unit1.Em2.ControlNodes".semiAutoSplice.jobs,
              jobStatus => "Unit1.EmNodes".emRelations.em02.sequence.Spare1.selectJobStatus[24]);
END_REGION

REGION Network 41: Select Job [25] Btm to Top : TAPPING
   RUNG wire#powerrail
      #instJob25(interlock := wire#w1, startCondition := wire#w2, parentReferenceDesignator := "Unit1.Em2.Config".em.referenceDesignator.combined, jobNumber := "U1EM2_JOB25", singleCycleJob := TRUE, hmiInterface := "Unit1.Em2.HmiInterface".semiAutoSplice.jobs, jobs := "Unit1.Em2.ControlNodes".semiAutoSplice.jobs, jobStatus => "Unit1.EmNodes".emRelations.em02.sequence.Spare1.selectJobStatus[25])
   END_RUNG
   RUNG wire#powerrail
      I_Contact( "Unit1.Em2.Alarms".emAlarms.error )
   END_RUNG wire#w1
   RUNG wire#powerrail
      Contact( #statUnitStatus.mode.production )
      Contact( #statUnitStatus.state.execute )
      Contact( "Unit1.EmNodes".emRelations.em02.sequence.Spare1.selectJobStatus[24].completed )
   END_RUNG wire#w2
   // the same network as SCL:
   #instJob25(parentReferenceDesignator := "Unit1.Em2.Config".em.referenceDesignator.combined,   // "LAF_SelectJob"
              jobNumber := "U1EM2_JOB25",
              singleCycleJob := TRUE,
              interlock := NOT "Unit1.Em2.Alarms".emAlarms.error,
              startCondition := #statUnitStatus.mode.production AND #statUnitStatus.state.execute AND "Unit1.EmNodes".emRelations.em02.sequence.Spare1.selectJobStatus[24].completed,
              hmiInterface := "Unit1.Em2.HmiInterface".semiAutoSplice.jobs,
              jobs := "Unit1.Em2.ControlNodes".semiAutoSplice.jobs,
              jobStatus => "Unit1.EmNodes".emRelations.em02.sequence.Spare1.selectJobStatus[25]);
END_REGION

REGION Network 42: Select Job [26] Btm to Top : Head Rotate Top (BWD)
   RUNG wire#powerrail
      #instJob26(interlock := wire#w1, startCondition := wire#w2, parentReferenceDesignator := "Unit1.Em2.Config".em.referenceDesignator.combined, jobNumber := "U1EM2_JOB26", singleCycleJob := TRUE, hmiInterface := "Unit1.Em2.HmiInterface".semiAutoSplice.jobs, jobs := "Unit1.Em2.ControlNodes".semiAutoSplice.jobs, jobStatus => "Unit1.EmNodes".emRelations.em02.sequence.Spare1.selectJobStatus[26])
   END_RUNG
   RUNG wire#powerrail
      I_Contact( "Unit1.Em2.Alarms".emAlarms.error )
   END_RUNG wire#w1
   RUNG wire#powerrail
      Contact( #statUnitStatus.mode.production )
      Contact( #statUnitStatus.state.execute )
      Contact( "Unit1.EmNodes".emRelations.em02.sequence.Spare1.selectJobStatus[25].completed )
   END_RUNG wire#w2
   // the same network as SCL:
   #instJob26(parentReferenceDesignator := "Unit1.Em2.Config".em.referenceDesignator.combined,   // "LAF_SelectJob"
              jobNumber := "U1EM2_JOB26",
              singleCycleJob := TRUE,
              interlock := NOT "Unit1.Em2.Alarms".emAlarms.error,
              startCondition := #statUnitStatus.mode.production AND #statUnitStatus.state.execute AND "Unit1.EmNodes".emRelations.em02.sequence.Spare1.selectJobStatus[25].completed,
              hmiInterface := "Unit1.Em2.HmiInterface".semiAutoSplice.jobs,
              jobs := "Unit1.Em2.ControlNodes".semiAutoSplice.jobs,
              jobStatus => "Unit1.EmNodes".emRelations.em02.sequence.Spare1.selectJobStatus[26]);
END_REGION

REGION Network 43: Select Job [27] Btm to Top : Pad Top/Btm Vacc Off & Pad Top/Btm Home (Down)
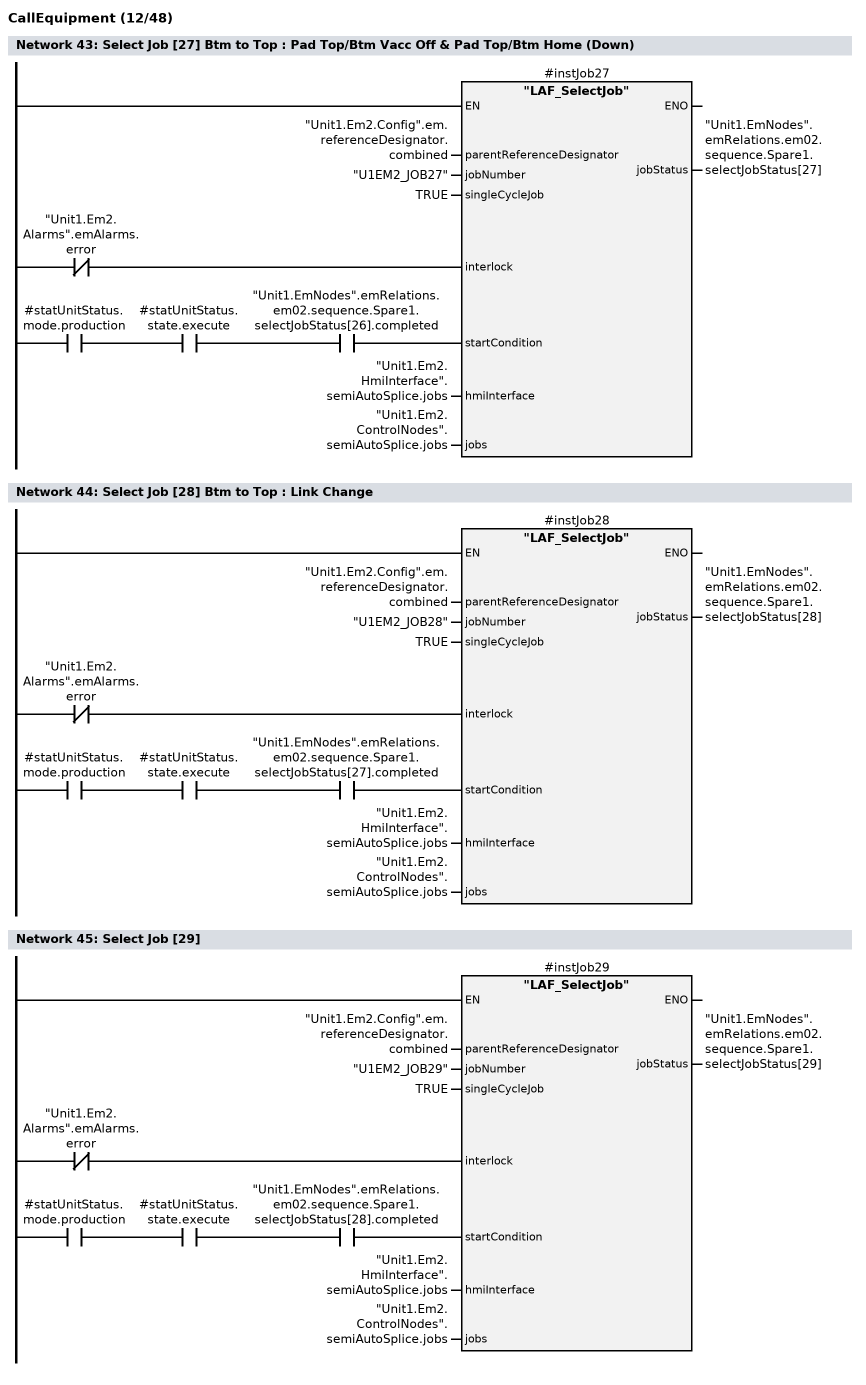
   RUNG wire#powerrail
      #instJob27(interlock := wire#w1, startCondition := wire#w2, parentReferenceDesignator := "Unit1.Em2.Config".em.referenceDesignator.combined, jobNumber := "U1EM2_JOB27", singleCycleJob := TRUE, hmiInterface := "Unit1.Em2.HmiInterface".semiAutoSplice.jobs, jobs := "Unit1.Em2.ControlNodes".semiAutoSplice.jobs, jobStatus => "Unit1.EmNodes".emRelations.em02.sequence.Spare1.selectJobStatus[27])
   END_RUNG
   RUNG wire#powerrail
      I_Contact( "Unit1.Em2.Alarms".emAlarms.error )
   END_RUNG wire#w1
   RUNG wire#powerrail
      Contact( #statUnitStatus.mode.production )
      Contact( #statUnitStatus.state.execute )
      Contact( "Unit1.EmNodes".emRelations.em02.sequence.Spare1.selectJobStatus[26].completed )
   END_RUNG wire#w2
   // the same network as SCL:
   #instJob27(parentReferenceDesignator := "Unit1.Em2.Config".em.referenceDesignator.combined,   // "LAF_SelectJob"
              jobNumber := "U1EM2_JOB27",
              singleCycleJob := TRUE,
              interlock := NOT "Unit1.Em2.Alarms".emAlarms.error,
              startCondition := #statUnitStatus.mode.production AND #statUnitStatus.state.execute AND "Unit1.EmNodes".emRelations.em02.sequence.Spare1.selectJobStatus[26].completed,
              hmiInterface := "Unit1.Em2.HmiInterface".semiAutoSplice.jobs,
              jobs := "Unit1.Em2.ControlNodes".semiAutoSplice.jobs,
              jobStatus => "Unit1.EmNodes".emRelations.em02.sequence.Spare1.selectJobStatus[27]);
END_REGION

REGION Network 44: Select Job [28] Btm to Top : Link Change
   RUNG wire#powerrail
      #instJob28(interlock := wire#w1, startCondition := wire#w2, parentReferenceDesignator := "Unit1.Em2.Config".em.referenceDesignator.combined, jobNumber := "U1EM2_JOB28", singleCycleJob := TRUE, hmiInterface := "Unit1.Em2.HmiInterface".semiAutoSplice.jobs, jobs := "Unit1.Em2.ControlNodes".semiAutoSplice.jobs, jobStatus => "Unit1.EmNodes".emRelations.em02.sequence.Spare1.selectJobStatus[28])
   END_RUNG
   RUNG wire#powerrail
      I_Contact( "Unit1.Em2.Alarms".emAlarms.error )
   END_RUNG wire#w1
   RUNG wire#powerrail
      Contact( #statUnitStatus.mode.production )
      Contact( #statUnitStatus.state.execute )
      Contact( "Unit1.EmNodes".emRelations.em02.sequence.Spare1.selectJobStatus[27].completed )
   END_RUNG wire#w2
   // the same network as SCL:
   #instJob28(parentReferenceDesignator := "Unit1.Em2.Config".em.referenceDesignator.combined,   // "LAF_SelectJob"
              jobNumber := "U1EM2_JOB28",
              singleCycleJob := TRUE,
              interlock := NOT "Unit1.Em2.Alarms".emAlarms.error,
              startCondition := #statUnitStatus.mode.production AND #statUnitStatus.state.execute AND "Unit1.EmNodes".emRelations.em02.sequence.Spare1.selectJobStatus[27].completed,
              hmiInterface := "Unit1.Em2.HmiInterface".semiAutoSplice.jobs,
              jobs := "Unit1.Em2.ControlNodes".semiAutoSplice.jobs,
              jobStatus => "Unit1.EmNodes".emRelations.em02.sequence.Spare1.selectJobStatus[28]);
END_REGION

REGION Network 45: Select Job [29]
   RUNG wire#powerrail
      #instJob29(interlock := wire#w1, startCondition := wire#w2, parentReferenceDesignator := "Unit1.Em2.Config".em.referenceDesignator.combined, jobNumber := "U1EM2_JOB29", singleCycleJob := TRUE, hmiInterface := "Unit1.Em2.HmiInterface".semiAutoSplice.jobs, jobs := "Unit1.Em2.ControlNodes".semiAutoSplice.jobs, jobStatus => "Unit1.EmNodes".emRelations.em02.sequence.Spare1.selectJobStatus[29])
   END_RUNG
   RUNG wire#powerrail
      I_Contact( "Unit1.Em2.Alarms".emAlarms.error )
   END_RUNG wire#w1
   RUNG wire#powerrail
      Contact( #statUnitStatus.mode.production )
      Contact( #statUnitStatus.state.execute )
      Contact( "Unit1.EmNodes".emRelations.em02.sequence.Spare1.selectJobStatus[28].completed )
   END_RUNG wire#w2
   // the same network as SCL:
   #instJob29(parentReferenceDesignator := "Unit1.Em2.Config".em.referenceDesignator.combined,   // "LAF_SelectJob"
              jobNumber := "U1EM2_JOB29",
              singleCycleJob := TRUE,
              interlock := NOT "Unit1.Em2.Alarms".emAlarms.error,
              startCondition := #statUnitStatus.mode.production AND #statUnitStatus.state.execute AND "Unit1.EmNodes".emRelations.em02.sequence.Spare1.selectJobStatus[28].completed,
              hmiInterface := "Unit1.Em2.HmiInterface".semiAutoSplice.jobs,
              jobs := "Unit1.Em2.ControlNodes".semiAutoSplice.jobs,
              jobStatus => "Unit1.EmNodes".emRelations.em02.sequence.Spare1.selectJobStatus[29]);
END_REGION

REGION Network 46: Select Job [30] FULL AUTO
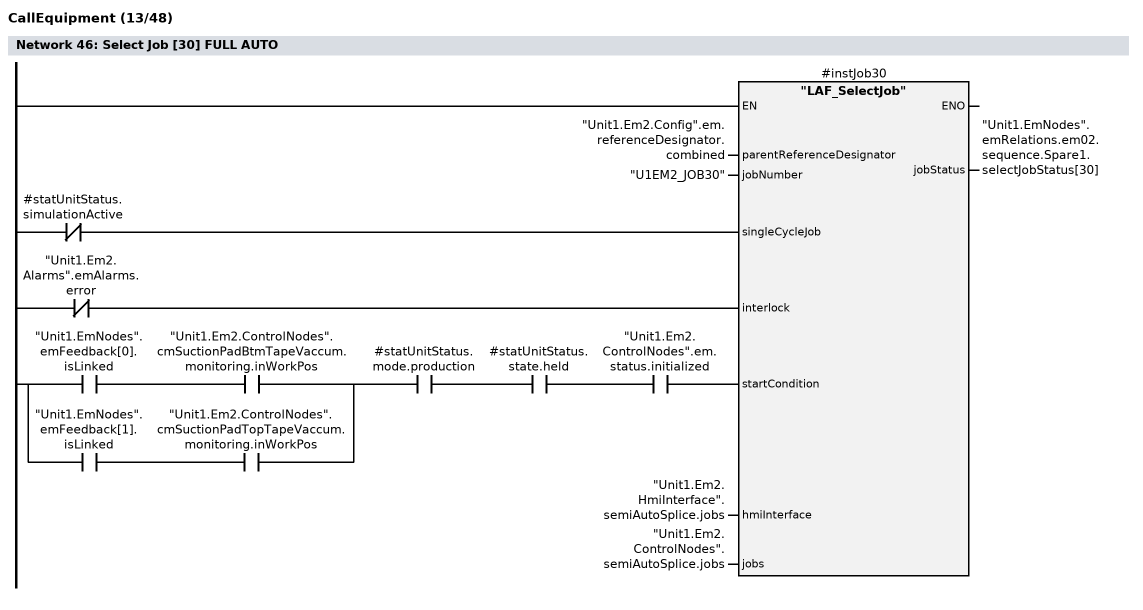
   RUNG wire#powerrail
      #instJob30(singleCycleJob := wire#w1, interlock := wire#w2, startCondition := wire#w4, parentReferenceDesignator := "Unit1.Em2.Config".em.referenceDesignator.combined, jobNumber := "U1EM2_JOB30", hmiInterface := "Unit1.Em2.HmiInterface".semiAutoSplice.jobs, jobs := "Unit1.Em2.ControlNodes".semiAutoSplice.jobs, jobStatus => "Unit1.EmNodes".emRelations.em02.sequence.Spare1.selectJobStatus[30])
   END_RUNG
   RUNG wire#powerrail
      I_Contact( #statUnitStatus.simulationActive )
   END_RUNG wire#w1
   RUNG wire#powerrail
      I_Contact( "Unit1.Em2.Alarms".emAlarms.error )
   END_RUNG wire#w2
   RUNG wire#powerrail
      Contact( "Unit1.EmNodes".emFeedback[0].isLinked )
      Contact( "Unit1.Em2.ControlNodes".cmSuctionPadBtmTapeVaccum.monitoring.inWorkPos )
      wire#w3
      Contact( #statUnitStatus.mode.production )
      Contact( #statUnitStatus.state.held )
      Contact( "Unit1.Em2.ControlNodes".em.status.initialized )
   END_RUNG wire#w4
   RUNG wire#powerrail
      Contact( "Unit1.EmNodes".emFeedback[1].isLinked )
      Contact( "Unit1.Em2.ControlNodes".cmSuctionPadTopTapeVaccum.monitoring.inWorkPos )
   END_RUNG wire#w3
   // the same network as SCL:
   #instJob30(parentReferenceDesignator := "Unit1.Em2.Config".em.referenceDesignator.combined,   // "LAF_SelectJob"
              jobNumber := "U1EM2_JOB30",
              singleCycleJob := NOT #statUnitStatus.simulationActive,
              interlock := NOT "Unit1.Em2.Alarms".emAlarms.error,
              startCondition := (("Unit1.EmNodes".emFeedback[0].isLinked AND "Unit1.Em2.ControlNodes".cmSuctionPadBtmTapeVaccum.monitoring.inWorkPos) OR ("Unit1.EmNodes".emFeedback[1].isLinked AND "Unit1.Em2.ControlNodes".cmSuctionPadTopTapeVaccum.monitoring.inWorkPos)) AND #statUnitStatus.mode.production AND #statUnitStatus.state.held AND "Unit1.Em2.ControlNodes".em.status.initialized,
              hmiInterface := "Unit1.Em2.HmiInterface".semiAutoSplice.jobs,
              jobs := "Unit1.Em2.ControlNodes".semiAutoSplice.jobs,
              jobStatus => "Unit1.EmNodes".emRelations.em02.sequence.Spare1.selectJobStatus[30]);
END_REGION

REGION Network 48: [SemiAutoSplice] Job Interface Request
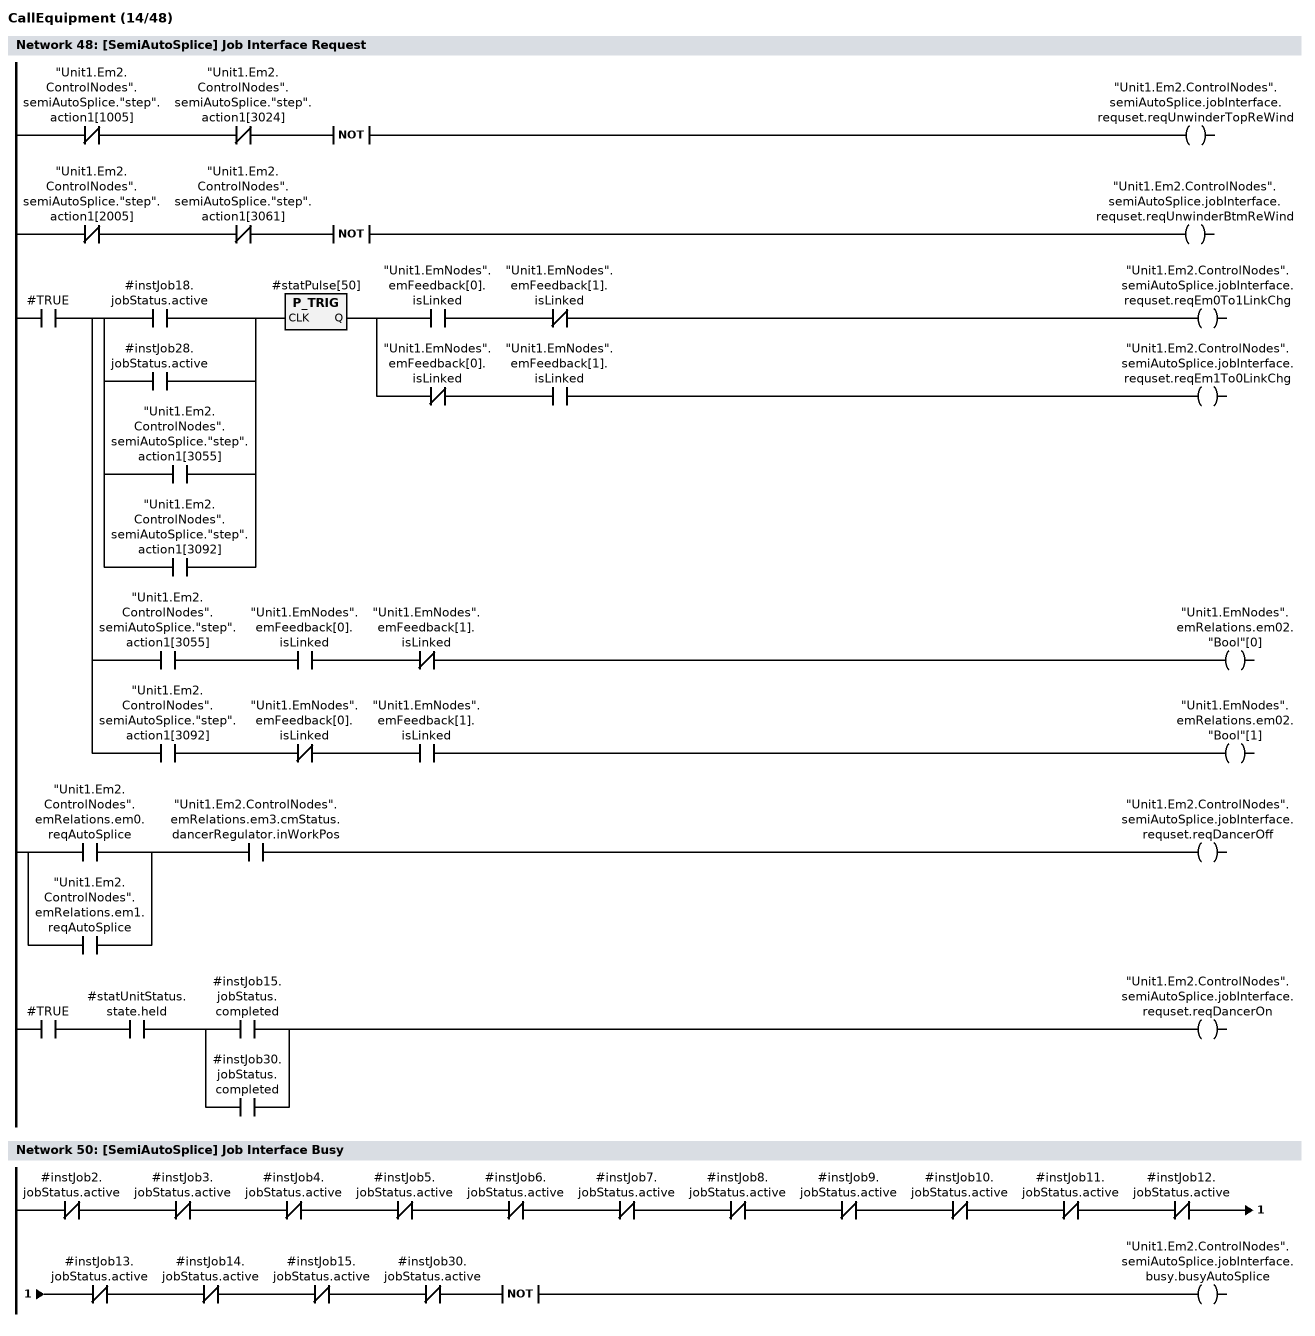
   RUNG wire#powerrail
      I_Contact( "Unit1.Em2.ControlNodes".semiAutoSplice."step".action1[1005] )
      I_Contact( "Unit1.Em2.ControlNodes".semiAutoSplice."step".action1[3024] )
      Not()
      Coil( "Unit1.Em2.ControlNodes".semiAutoSplice.jobInterface.requset.reqUnwinderTopReWind )
   END_RUNG
   RUNG wire#powerrail
      I_Contact( "Unit1.Em2.ControlNodes".semiAutoSplice."step".action1[2005] )
      I_Contact( "Unit1.Em2.ControlNodes".semiAutoSplice."step".action1[3061] )
      Not()
      Coil( "Unit1.Em2.ControlNodes".semiAutoSplice.jobInterface.requset.reqUnwinderBtmReWind )
   END_RUNG
   RUNG wire#powerrail
      Contact( #TRUE )
      wire#w1
      Contact( #instJob18.jobStatus.active )
      wire#w2
      P_Trig( #statPulse[50] )
      wire#w3
      Contact( "Unit1.EmNodes".emFeedback[0].isLinked )
      I_Contact( "Unit1.EmNodes".emFeedback[1].isLinked )
      Coil( "Unit1.Em2.ControlNodes".semiAutoSplice.jobInterface.requset.reqEm0To1LinkChg )
   END_RUNG
   RUNG wire#w1
      Contact( #instJob28.jobStatus.active )
   END_RUNG wire#w2
   RUNG wire#w1
      Contact( "Unit1.Em2.ControlNodes".semiAutoSplice."step".action1[3055] )
   END_RUNG wire#w2
   RUNG wire#w1
      Contact( "Unit1.Em2.ControlNodes".semiAutoSplice."step".action1[3092] )
   END_RUNG wire#w2
   RUNG wire#w3
      I_Contact( "Unit1.EmNodes".emFeedback[0].isLinked )
      Contact( "Unit1.EmNodes".emFeedback[1].isLinked )
      Coil( "Unit1.Em2.ControlNodes".semiAutoSplice.jobInterface.requset.reqEm1To0LinkChg )
   END_RUNG
   RUNG wire#w1
      Contact( "Unit1.Em2.ControlNodes".semiAutoSplice."step".action1[3055] )
      Contact( "Unit1.EmNodes".emFeedback[0].isLinked )
      I_Contact( "Unit1.EmNodes".emFeedback[1].isLinked )
      Coil( "Unit1.EmNodes".emRelations.em02."Bool"[0] )
   END_RUNG
   RUNG wire#w1
      Contact( "Unit1.Em2.ControlNodes".semiAutoSplice."step".action1[3092] )
      I_Contact( "Unit1.EmNodes".emFeedback[0].isLinked )
      Contact( "Unit1.EmNodes".emFeedback[1].isLinked )
      Coil( "Unit1.EmNodes".emRelations.em02."Bool"[1] )
   END_RUNG
   RUNG wire#powerrail
      Contact( "Unit1.Em2.ControlNodes".emRelations.em0.reqAutoSplice )
      wire#w4
      Contact( "Unit1.Em2.ControlNodes".emRelations.em3.cmStatus.dancerRegulator.inWorkPos )
      Coil( "Unit1.Em2.ControlNodes".semiAutoSplice.jobInterface.requset.reqDancerOff )
   END_RUNG
   RUNG wire#powerrail
      Contact( "Unit1.Em2.ControlNodes".emRelations.em1.reqAutoSplice )
   END_RUNG wire#w4
   RUNG wire#powerrail
      Contact( #TRUE )
      Contact( #statUnitStatus.state.held )
      wire#w5
      Contact( #instJob15.jobStatus.completed )
      wire#w6
      Coil( "Unit1.Em2.ControlNodes".semiAutoSplice.jobInterface.requset.reqDancerOn )
   END_RUNG
   RUNG wire#w5
      Contact( #instJob30.jobStatus.completed )
   END_RUNG wire#w6
   // the same network as SCL:
   "Unit1.Em2.ControlNodes".semiAutoSplice.jobInterface.requset.reqUnwinderTopReWind := NOT (NOT "Unit1.Em2.ControlNodes".semiAutoSplice."step".action1[1005] AND NOT "Unit1.Em2.ControlNodes".semiAutoSplice."step".action1[3024]);
   "Unit1.Em2.ControlNodes".semiAutoSplice.jobInterface.requset.reqUnwinderBtmReWind := NOT (NOT "Unit1.Em2.ControlNodes".semiAutoSplice."step".action1[2005] AND NOT "Unit1.Em2.ControlNodes".semiAutoSplice."step".action1[3061]);
   #_w1 := #TRUE AND (#instJob18.jobStatus.active OR #instJob28.jobStatus.active OR "Unit1.Em2.ControlNodes".semiAutoSplice."step".action1[3055] OR "Unit1.Em2.ControlNodes".semiAutoSplice."step".action1[3092]);
   #_w2 := #_w1 AND NOT #statPulse[50];   // rising edge
   #statPulse[50] := #_w1;
   "Unit1.Em2.ControlNodes".semiAutoSplice.jobInterface.requset.reqEm0To1LinkChg := #_w2 AND "Unit1.EmNodes".emFeedback[0].isLinked AND NOT "Unit1.EmNodes".emFeedback[1].isLinked;
   "Unit1.Em2.ControlNodes".semiAutoSplice.jobInterface.requset.reqEm1To0LinkChg := #_w2 AND NOT "Unit1.EmNodes".emFeedback[0].isLinked AND "Unit1.EmNodes".emFeedback[1].isLinked;
   "Unit1.EmNodes".emRelations.em02."Bool"[0] := #TRUE AND "Unit1.Em2.ControlNodes".semiAutoSplice."step".action1[3055] AND "Unit1.EmNodes".emFeedback[0].isLinked AND NOT "Unit1.EmNodes".emFeedback[1].isLinked;
   "Unit1.EmNodes".emRelations.em02."Bool"[1] := #TRUE AND "Unit1.Em2.ControlNodes".semiAutoSplice."step".action1[3092] AND NOT "Unit1.EmNodes".emFeedback[0].isLinked AND "Unit1.EmNodes".emFeedback[1].isLinked;
   "Unit1.Em2.ControlNodes".semiAutoSplice.jobInterface.requset.reqDancerOff := ("Unit1.Em2.ControlNodes".emRelations.em0.reqAutoSplice OR "Unit1.Em2.ControlNodes".emRelations.em1.reqAutoSplice) AND "Unit1.Em2.ControlNodes".emRelations.em3.cmStatus.dancerRegulator.inWorkPos;
   "Unit1.Em2.ControlNodes".semiAutoSplice.jobInterface.requset.reqDancerOn := #TRUE AND #statUnitStatus.state.held AND (#instJob15.jobStatus.completed OR #instJob30.jobStatus.completed);
END_REGION

REGION Network 49: [SemiAutoSplice] Job Interface Ready
END_REGION

REGION Network 50: [SemiAutoSplice] Job Interface Busy
   RUNG wire#powerrail
      I_Contact( #instJob2.jobStatus.active )
      I_Contact( #instJob3.jobStatus.active )
      I_Contact( #instJob4.jobStatus.active )
      I_Contact( #instJob5.jobStatus.active )
      I_Contact( #instJob6.jobStatus.active )
      I_Contact( #instJob7.jobStatus.active )
      I_Contact( #instJob8.jobStatus.active )
      I_Contact( #instJob9.jobStatus.active )
      I_Contact( #instJob10.jobStatus.active )
      I_Contact( #instJob11.jobStatus.active )
      I_Contact( #instJob12.jobStatus.active )
      I_Contact( #instJob13.jobStatus.active )
      I_Contact( #instJob14.jobStatus.active )
      I_Contact( #instJob15.jobStatus.active )
      I_Contact( #instJob30.jobStatus.active )
      Not()
      Coil( "Unit1.Em2.ControlNodes".semiAutoSplice.jobInterface.busy.busyAutoSplice )
   END_RUNG
   // the same network as SCL:
   "Unit1.Em2.ControlNodes".semiAutoSplice.jobInterface.busy.busyAutoSplice := NOT (NOT #instJob2.jobStatus.active AND NOT #instJob3.jobStatus.active AND NOT #instJob4.jobStatus.active AND NOT #instJob5.jobStatus.active AND NOT #instJob6.jobStatus.active AND NOT #instJob7.jobStatus.active AND NOT #instJob8.jobStatus.active AND NOT #instJob9.jobStatus.active AND NOT #instJob10.jobStatus.active AND NOT #instJob11.jobStatus.active AND NOT #instJob12.jobStatus.active AND NOT #instJob13.jobStatus.active AND NOT #instJob14.jobStatus.active AND NOT #instJob15.jobStatus.active AND NOT #instJob30.jobStatus.active);
END_REGION

REGION Network 51: [SemiAutoSplice] Job Interface Done
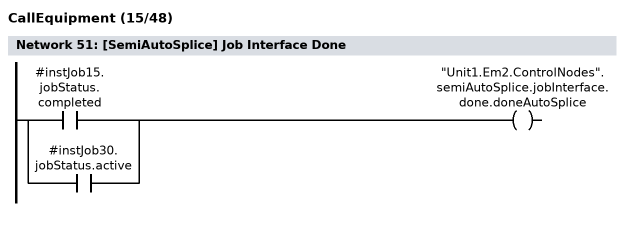
   RUNG wire#powerrail
      Contact( #instJob15.jobStatus.completed )
      wire#w1
      Coil( "Unit1.Em2.ControlNodes".semiAutoSplice.jobInterface.done.doneAutoSplice )
   END_RUNG
   RUNG wire#powerrail
      Contact( #instJob30.jobStatus.active )
   END_RUNG wire#w1
   // the same network as SCL:
   "Unit1.Em2.ControlNodes".semiAutoSplice.jobInterface.done.doneAutoSplice := #instJob15.jobStatus.completed OR #instJob30.jobStatus.active;
END_REGION

REGION Network 52: [SemiAutoSplice] Job Working Done
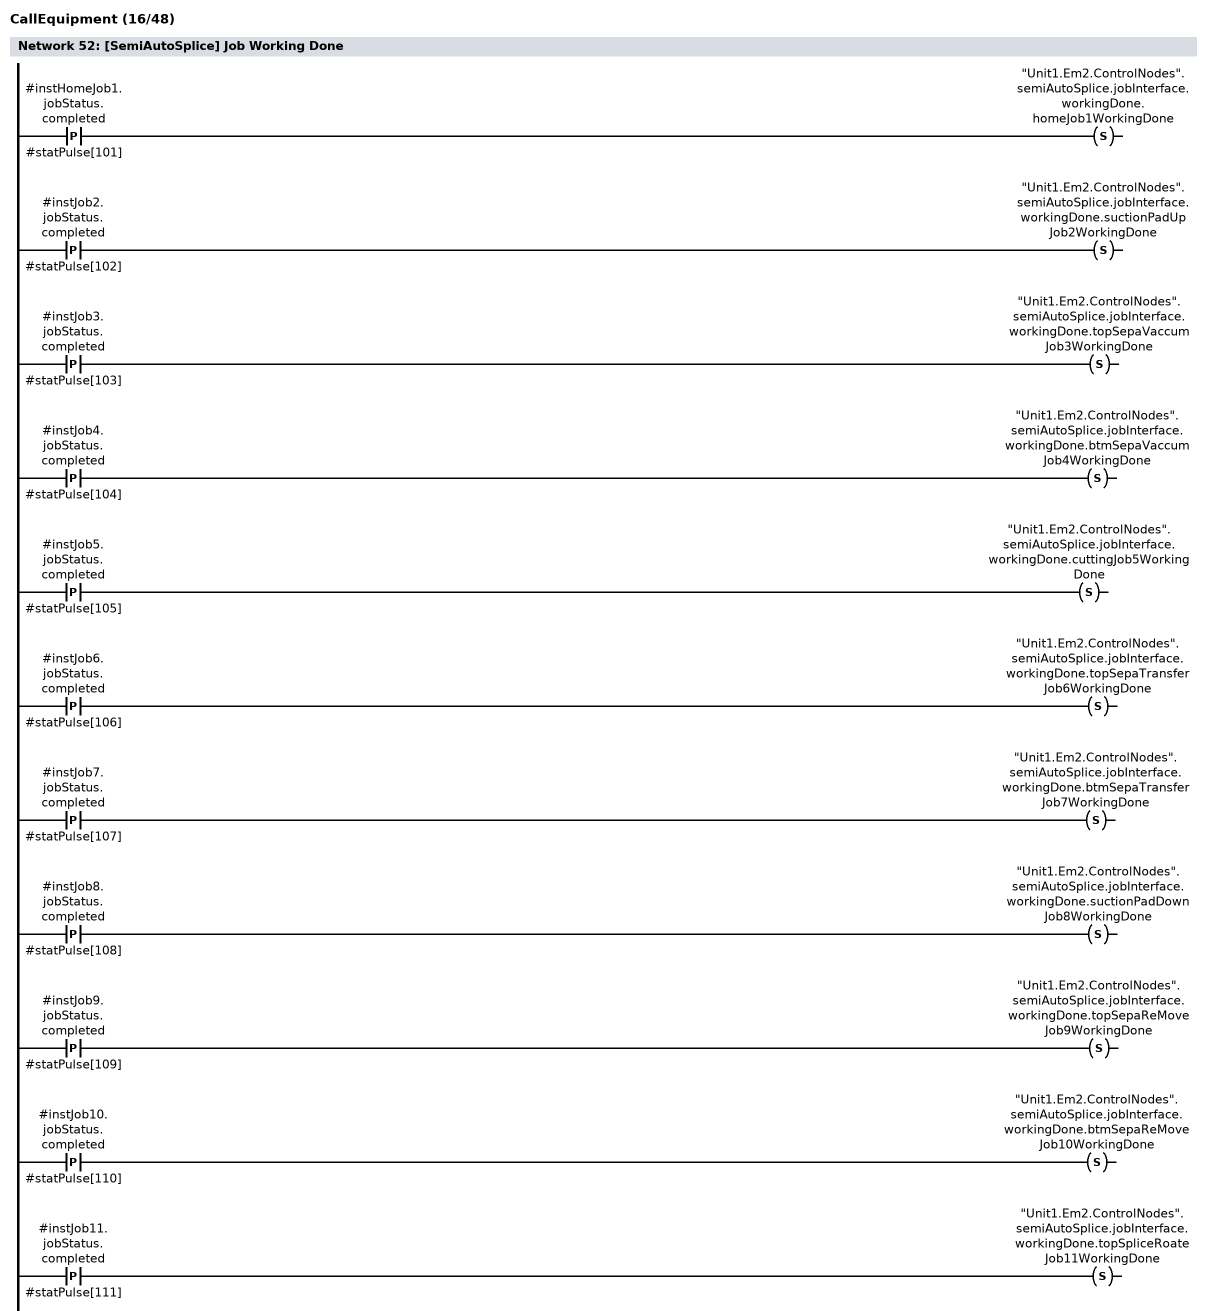
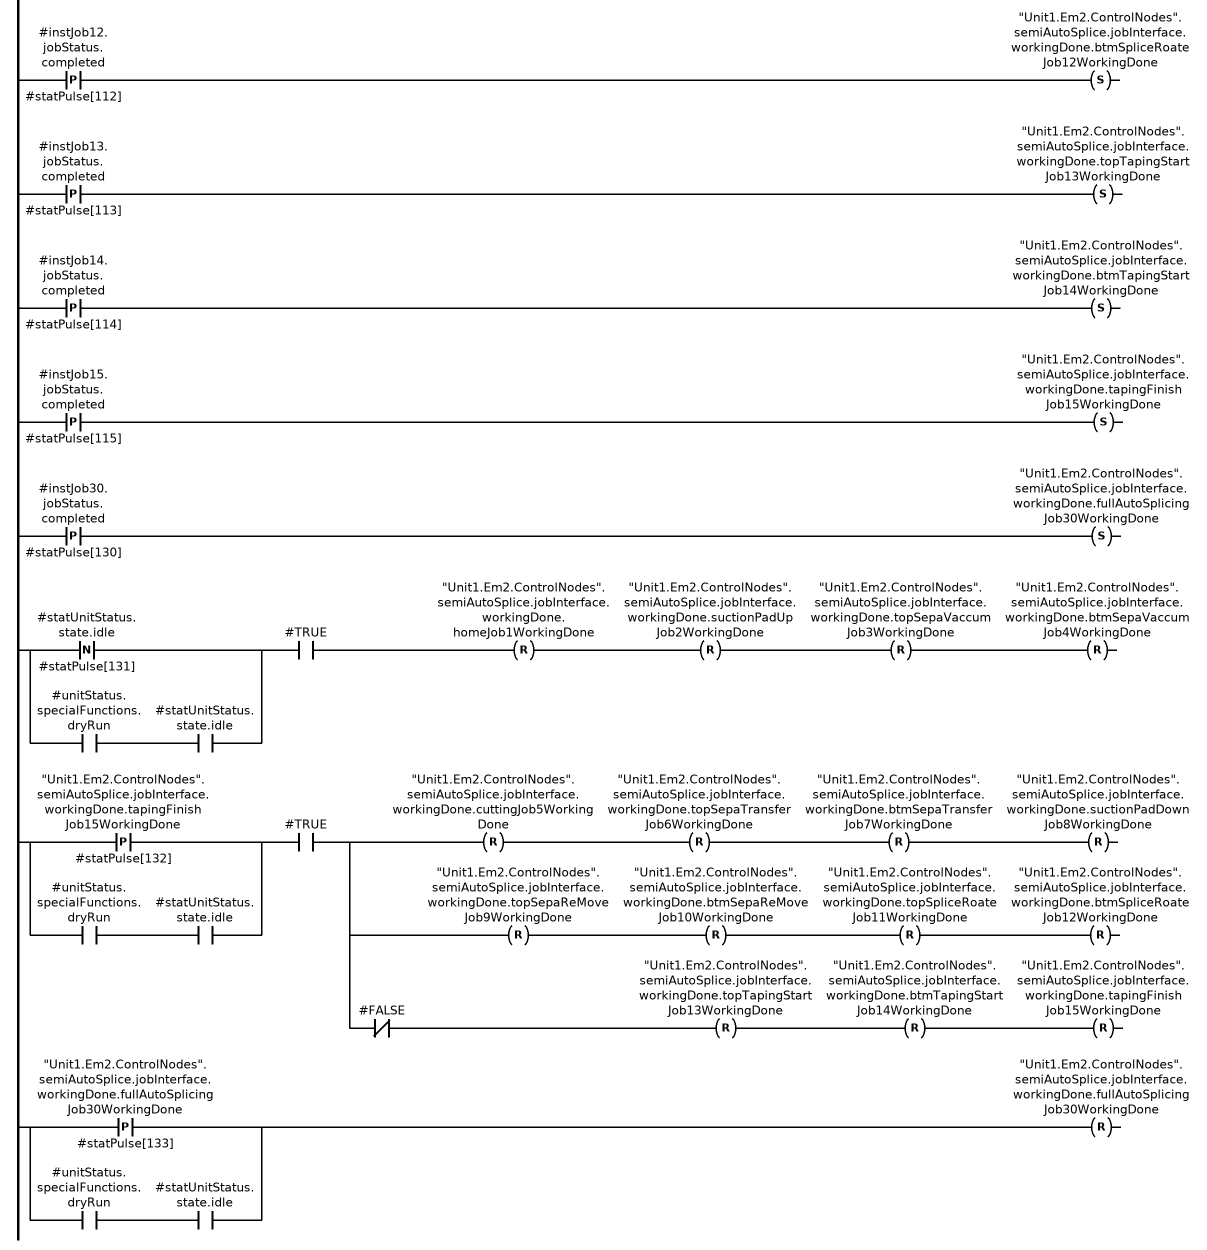
   RUNG wire#powerrail
      P_Contact(operand := #instHomeJob1.jobStatus.completed, bit := #statPulse[101])
      S_Coil( "Unit1.Em2.ControlNodes".semiAutoSplice.jobInterface.workingDone.homeJob1WorkingDone )
   END_RUNG
   RUNG wire#powerrail
      P_Contact(operand := #instJob2.jobStatus.completed, bit := #statPulse[102])
      S_Coil( "Unit1.Em2.ControlNodes".semiAutoSplice.jobInterface.workingDone.suctionPadUpJob2WorkingDone )
   END_RUNG
   RUNG wire#powerrail
      P_Contact(operand := #instJob3.jobStatus.completed, bit := #statPulse[103])
      S_Coil( "Unit1.Em2.ControlNodes".semiAutoSplice.jobInterface.workingDone.topSepaVaccumJob3WorkingDone )
   END_RUNG
   RUNG wire#powerrail
      P_Contact(operand := #instJob4.jobStatus.completed, bit := #statPulse[104])
      S_Coil( "Unit1.Em2.ControlNodes".semiAutoSplice.jobInterface.workingDone.btmSepaVaccumJob4WorkingDone )
   END_RUNG
   RUNG wire#powerrail
      P_Contact(operand := #instJob5.jobStatus.completed, bit := #statPulse[105])
      S_Coil( "Unit1.Em2.ControlNodes".semiAutoSplice.jobInterface.workingDone.cuttingJob5WorkingDone )
   END_RUNG
   RUNG wire#powerrail
      P_Contact(operand := #instJob6.jobStatus.completed, bit := #statPulse[106])
      S_Coil( "Unit1.Em2.ControlNodes".semiAutoSplice.jobInterface.workingDone.topSepaTransferJob6WorkingDone )
   END_RUNG
   RUNG wire#powerrail
      P_Contact(operand := #instJob7.jobStatus.completed, bit := #statPulse[107])
      S_Coil( "Unit1.Em2.ControlNodes".semiAutoSplice.jobInterface.workingDone.btmSepaTransferJob7WorkingDone )
   END_RUNG
   RUNG wire#powerrail
      P_Contact(operand := #instJob8.jobStatus.completed, bit := #statPulse[108])
      S_Coil( "Unit1.Em2.ControlNodes".semiAutoSplice.jobInterface.workingDone.suctionPadDownJob8WorkingDone )
   END_RUNG
   RUNG wire#powerrail
      P_Contact(operand := #instJob9.jobStatus.completed, bit := #statPulse[109])
      S_Coil( "Unit1.Em2.ControlNodes".semiAutoSplice.jobInterface.workingDone.topSepaReMoveJob9WorkingDone )
   END_RUNG
   RUNG wire#powerrail
      P_Contact(operand := #instJob10.jobStatus.completed, bit := #statPulse[110])
      S_Coil( "Unit1.Em2.ControlNodes".semiAutoSplice.jobInterface.workingDone.btmSepaReMoveJob10WorkingDone )
   END_RUNG
   RUNG wire#powerrail
      P_Contact(operand := #instJob11.jobStatus.completed, bit := #statPulse[111])
      S_Coil( "Unit1.Em2.ControlNodes".semiAutoSplice.jobInterface.workingDone.topSpliceRoateJob11WorkingDone )
   END_RUNG
   RUNG wire#powerrail
      P_Contact(operand := #instJob12.jobStatus.completed, bit := #statPulse[112])
      S_Coil( "Unit1.Em2.ControlNodes".semiAutoSplice.jobInterface.workingDone.btmSpliceRoateJob12WorkingDone )
   END_RUNG
   RUNG wire#powerrail
      P_Contact(operand := #instJob13.jobStatus.completed, bit := #statPulse[113])
      S_Coil( "Unit1.Em2.ControlNodes".semiAutoSplice.jobInterface.workingDone.topTapingStartJob13WorkingDone )
   END_RUNG
   RUNG wire#powerrail
      P_Contact(operand := #instJob14.jobStatus.completed, bit := #statPulse[114])
      S_Coil( "Unit1.Em2.ControlNodes".semiAutoSplice.jobInterface.workingDone.btmTapingStartJob14WorkingDone )
   END_RUNG
   RUNG wire#powerrail
      P_Contact(operand := #instJob15.jobStatus.completed, bit := #statPulse[115])
      S_Coil( "Unit1.Em2.ControlNodes".semiAutoSplice.jobInterface.workingDone.tapingFinishJob15WorkingDone )
   END_RUNG
   RUNG wire#powerrail
      P_Contact(operand := #instJob30.jobStatus.completed, bit := #statPulse[130])
      S_Coil( "Unit1.Em2.ControlNodes".semiAutoSplice.jobInterface.workingDone.fullAutoSplicingJob30WorkingDone )
   END_RUNG
   RUNG wire#powerrail
      N_Contact(operand := #statUnitStatus.state.idle, bit := #statPulse[131])
      wire#w1
      Contact( #TRUE )
      R_Coil( "Unit1.Em2.ControlNodes".semiAutoSplice.jobInterface.workingDone.homeJob1WorkingDone )
      R_Coil( "Unit1.Em2.ControlNodes".semiAutoSplice.jobInterface.workingDone.suctionPadUpJob2WorkingDone )
      R_Coil( "Unit1.Em2.ControlNodes".semiAutoSplice.jobInterface.workingDone.topSepaVaccumJob3WorkingDone )
      R_Coil( "Unit1.Em2.ControlNodes".semiAutoSplice.jobInterface.workingDone.btmSepaVaccumJob4WorkingDone )
   END_RUNG
   RUNG wire#powerrail
      Contact( #unitStatus.specialFunctions.dryRun )
      Contact( #statUnitStatus.state.idle )
   END_RUNG wire#w1
   RUNG wire#powerrail
      P_Contact(operand := "Unit1.Em2.ControlNodes".semiAutoSplice.jobInterface.workingDone.tapingFinishJob15WorkingDone, bit := #statPulse[132])
      wire#w2
      Contact( #TRUE )
      wire#w3
      R_Coil( "Unit1.Em2.ControlNodes".semiAutoSplice.jobInterface.workingDone.cuttingJob5WorkingDone )
      R_Coil( "Unit1.Em2.ControlNodes".semiAutoSplice.jobInterface.workingDone.topSepaTransferJob6WorkingDone )
      R_Coil( "Unit1.Em2.ControlNodes".semiAutoSplice.jobInterface.workingDone.btmSepaTransferJob7WorkingDone )
      R_Coil( "Unit1.Em2.ControlNodes".semiAutoSplice.jobInterface.workingDone.suctionPadDownJob8WorkingDone )
   END_RUNG
   RUNG wire#powerrail
      Contact( #unitStatus.specialFunctions.dryRun )
      Contact( #statUnitStatus.state.idle )
   END_RUNG wire#w2
   RUNG wire#w3
      R_Coil( "Unit1.Em2.ControlNodes".semiAutoSplice.jobInterface.workingDone.topSepaReMoveJob9WorkingDone )
      R_Coil( "Unit1.Em2.ControlNodes".semiAutoSplice.jobInterface.workingDone.btmSepaReMoveJob10WorkingDone )
      R_Coil( "Unit1.Em2.ControlNodes".semiAutoSplice.jobInterface.workingDone.topSpliceRoateJob11WorkingDone )
      R_Coil( "Unit1.Em2.ControlNodes".semiAutoSplice.jobInterface.workingDone.btmSpliceRoateJob12WorkingDone )
   END_RUNG
   RUNG wire#w3
      I_Contact( #FALSE )
      R_Coil( "Unit1.Em2.ControlNodes".semiAutoSplice.jobInterface.workingDone.topTapingStartJob13WorkingDone )
      R_Coil( "Unit1.Em2.ControlNodes".semiAutoSplice.jobInterface.workingDone.btmTapingStartJob14WorkingDone )
      R_Coil( "Unit1.Em2.ControlNodes".semiAutoSplice.jobInterface.workingDone.tapingFinishJob15WorkingDone )
   END_RUNG
   RUNG wire#powerrail
      P_Contact(operand := "Unit1.Em2.ControlNodes".semiAutoSplice.jobInterface.workingDone.fullAutoSplicingJob30WorkingDone, bit := #statPulse[133])
      wire#w4
      R_Coil( "Unit1.Em2.ControlNodes".semiAutoSplice.jobInterface.workingDone.fullAutoSplicingJob30WorkingDone )
   END_RUNG
   RUNG wire#powerrail
      Contact( #unitStatus.specialFunctions.dryRun )
      Contact( #statUnitStatus.state.idle )
   END_RUNG wire#w4
   // the same network as SCL:
   #_w1 := #instHomeJob1.jobStatus.completed AND NOT #statPulse[101];   // rising edge of #instHomeJob1.jobStatus.completed
   #statPulse[101] := #instHomeJob1.jobStatus.completed;
   IF #_w1 THEN
       "Unit1.Em2.ControlNodes".semiAutoSplice.jobInterface.workingDone.homeJob1WorkingDone := TRUE;
   END_IF;
   #_w2 := #instJob2.jobStatus.completed AND NOT #statPulse[102];   // rising edge of #instJob2.jobStatus.completed
   #statPulse[102] := #instJob2.jobStatus.completed;
   IF #_w2 THEN
       "Unit1.Em2.ControlNodes".semiAutoSplice.jobInterface.workingDone.suctionPadUpJob2WorkingDone := TRUE;
   END_IF;
   #_w3 := #instJob3.jobStatus.completed AND NOT #statPulse[103];   // rising edge of #instJob3.jobStatus.completed
   #statPulse[103] := #instJob3.jobStatus.completed;
   IF #_w3 THEN
       "Unit1.Em2.ControlNodes".semiAutoSplice.jobInterface.workingDone.topSepaVaccumJob3WorkingDone := TRUE;
   END_IF;
   #_w4 := #instJob4.jobStatus.completed AND NOT #statPulse[104];   // rising edge of #instJob4.jobStatus.completed
   #statPulse[104] := #instJob4.jobStatus.completed;
   IF #_w4 THEN
       "Unit1.Em2.ControlNodes".semiAutoSplice.jobInterface.workingDone.btmSepaVaccumJob4WorkingDone := TRUE;
   END_IF;
   #_w5 := #instJob5.jobStatus.completed AND NOT #statPulse[105];   // rising edge of #instJob5.jobStatus.completed
   #statPulse[105] := #instJob5.jobStatus.completed;
   IF #_w5 THEN
       "Unit1.Em2.ControlNodes".semiAutoSplice.jobInterface.workingDone.cuttingJob5WorkingDone := TRUE;
   END_IF;
   #_w6 := #instJob6.jobStatus.completed AND NOT #statPulse[106];   // rising edge of #instJob6.jobStatus.completed
   #statPulse[106] := #instJob6.jobStatus.completed;
   IF #_w6 THEN
       "Unit1.Em2.ControlNodes".semiAutoSplice.jobInterface.workingDone.topSepaTransferJob6WorkingDone := TRUE;
   END_IF;
   #_w7 := #instJob7.jobStatus.completed AND NOT #statPulse[107];   // rising edge of #instJob7.jobStatus.completed
   #statPulse[107] := #instJob7.jobStatus.completed;
   IF #_w7 THEN
       "Unit1.Em2.ControlNodes".semiAutoSplice.jobInterface.workingDone.btmSepaTransferJob7WorkingDone := TRUE;
   END_IF;
   #_w8 := #instJob8.jobStatus.completed AND NOT #statPulse[108];   // rising edge of #instJob8.jobStatus.completed
   #statPulse[108] := #instJob8.jobStatus.completed;
   IF #_w8 THEN
       "Unit1.Em2.ControlNodes".semiAutoSplice.jobInterface.workingDone.suctionPadDownJob8WorkingDone := TRUE;
   END_IF;
   #_w9 := #instJob9.jobStatus.completed AND NOT #statPulse[109];   // rising edge of #instJob9.jobStatus.completed
   #statPulse[109] := #instJob9.jobStatus.completed;
   IF #_w9 THEN
       "Unit1.Em2.ControlNodes".semiAutoSplice.jobInterface.workingDone.topSepaReMoveJob9WorkingDone := TRUE;
   END_IF;
   #_w10 := #instJob10.jobStatus.completed AND NOT #statPulse[110];   // rising edge of #instJob10.jobStatus.completed
   #statPulse[110] := #instJob10.jobStatus.completed;
   IF #_w10 THEN
       "Unit1.Em2.ControlNodes".semiAutoSplice.jobInterface.workingDone.btmSepaReMoveJob10WorkingDone := TRUE;
   END_IF;
   #_w11 := #instJob11.jobStatus.completed AND NOT #statPulse[111];   // rising edge of #instJob11.jobStatus.completed
   #statPulse[111] := #instJob11.jobStatus.completed;
   IF #_w11 THEN
       "Unit1.Em2.ControlNodes".semiAutoSplice.jobInterface.workingDone.topSpliceRoateJob11WorkingDone := TRUE;
   END_IF;
   #_w12 := #instJob12.jobStatus.completed AND NOT #statPulse[112];   // rising edge of #instJob12.jobStatus.completed
   #statPulse[112] := #instJob12.jobStatus.completed;
   IF #_w12 THEN
       "Unit1.Em2.ControlNodes".semiAutoSplice.jobInterface.workingDone.btmSpliceRoateJob12WorkingDone := TRUE;
   END_IF;
   #_w13 := #instJob13.jobStatus.completed AND NOT #statPulse[113];   // rising edge of #instJob13.jobStatus.completed
   #statPulse[113] := #instJob13.jobStatus.completed;
   IF #_w13 THEN
       "Unit1.Em2.ControlNodes".semiAutoSplice.jobInterface.workingDone.topTapingStartJob13WorkingDone := TRUE;
   END_IF;
   #_w14 := #instJob14.jobStatus.completed AND NOT #statPulse[114];   // rising edge of #instJob14.jobStatus.completed
   #statPulse[114] := #instJob14.jobStatus.completed;
   IF #_w14 THEN
       "Unit1.Em2.ControlNodes".semiAutoSplice.jobInterface.workingDone.btmTapingStartJob14WorkingDone := TRUE;
   END_IF;
   #_w15 := #instJob15.jobStatus.completed AND NOT #statPulse[115];   // rising edge of #instJob15.jobStatus.completed
   #statPulse[115] := #instJob15.jobStatus.completed;
   IF #_w15 THEN
       "Unit1.Em2.ControlNodes".semiAutoSplice.jobInterface.workingDone.tapingFinishJob15WorkingDone := TRUE;
   END_IF;
   #_w16 := #instJob30.jobStatus.completed AND NOT #statPulse[130];   // rising edge of #instJob30.jobStatus.completed
   #statPulse[130] := #instJob30.jobStatus.completed;
   IF #_w16 THEN
       "Unit1.Em2.ControlNodes".semiAutoSplice.jobInterface.workingDone.fullAutoSplicingJob30WorkingDone := TRUE;
   END_IF;
   #_w17 := NOT #statUnitStatus.state.idle AND #statPulse[131];   // falling edge of #statUnitStatus.state.idle
   #statPulse[131] := #statUnitStatus.state.idle;
   IF (#_w17 OR (#unitStatus.specialFunctions.dryRun AND #statUnitStatus.state.idle)) AND #TRUE THEN
       "Unit1.Em2.ControlNodes".semiAutoSplice.jobInterface.workingDone.homeJob1WorkingDone := FALSE;
       "Unit1.Em2.ControlNodes".semiAutoSplice.jobInterface.workingDone.suctionPadUpJob2WorkingDone := FALSE;
       "Unit1.Em2.ControlNodes".semiAutoSplice.jobInterface.workingDone.topSepaVaccumJob3WorkingDone := FALSE;
       "Unit1.Em2.ControlNodes".semiAutoSplice.jobInterface.workingDone.btmSepaVaccumJob4WorkingDone := FALSE;
   END_IF;
   #_w18 := "Unit1.Em2.ControlNodes".semiAutoSplice.jobInterface.workingDone.tapingFinishJob15WorkingDone AND NOT #statPulse[132];   // rising edge of "Unit1.Em2.ControlNodes".semiAutoSplice.jobInterface.workingDone.tapingFinishJob15WorkingDone
   #statPulse[132] := "Unit1.Em2.ControlNodes".semiAutoSplice.jobInterface.workingDone.tapingFinishJob15WorkingDone;
   #_w19 := (#_w18 OR (#unitStatus.specialFunctions.dryRun AND #statUnitStatus.state.idle)) AND #TRUE;
   IF #_w19 THEN
       "Unit1.Em2.ControlNodes".semiAutoSplice.jobInterface.workingDone.cuttingJob5WorkingDone := FALSE;
       "Unit1.Em2.ControlNodes".semiAutoSplice.jobInterface.workingDone.topSepaTransferJob6WorkingDone := FALSE;
       "Unit1.Em2.ControlNodes".semiAutoSplice.jobInterface.workingDone.btmSepaTransferJob7WorkingDone := FALSE;
       "Unit1.Em2.ControlNodes".semiAutoSplice.jobInterface.workingDone.suctionPadDownJob8WorkingDone := FALSE;
       "Unit1.Em2.ControlNodes".semiAutoSplice.jobInterface.workingDone.topSepaReMoveJob9WorkingDone := FALSE;
       "Unit1.Em2.ControlNodes".semiAutoSplice.jobInterface.workingDone.btmSepaReMoveJob10WorkingDone := FALSE;
       "Unit1.Em2.ControlNodes".semiAutoSplice.jobInterface.workingDone.topSpliceRoateJob11WorkingDone := FALSE;
       "Unit1.Em2.ControlNodes".semiAutoSplice.jobInterface.workingDone.btmSpliceRoateJob12WorkingDone := FALSE;
   END_IF;
   IF #_w19 AND NOT #FALSE THEN
       "Unit1.Em2.ControlNodes".semiAutoSplice.jobInterface.workingDone.topTapingStartJob13WorkingDone := FALSE;
       "Unit1.Em2.ControlNodes".semiAutoSplice.jobInterface.workingDone.btmTapingStartJob14WorkingDone := FALSE;
       "Unit1.Em2.ControlNodes".semiAutoSplice.jobInterface.workingDone.tapingFinishJob15WorkingDone := FALSE;
   END_IF;
   #_w20 := "Unit1.Em2.ControlNodes".semiAutoSplice.jobInterface.workingDone.fullAutoSplicingJob30WorkingDone AND NOT #statPulse[133];   // rising edge of "Unit1.Em2.ControlNodes".semiAutoSplice.jobInterface.workingDone.fullAutoSplicingJob30WorkingDone
   #statPulse[133] := "Unit1.Em2.ControlNodes".semiAutoSplice.jobInterface.workingDone.fullAutoSplicingJob30WorkingDone;
   IF #_w20 OR (#unitStatus.specialFunctions.dryRun AND #statUnitStatus.state.idle) THEN
       "Unit1.Em2.ControlNodes".semiAutoSplice.jobInterface.workingDone.fullAutoSplicingJob30WorkingDone := FALSE;
   END_IF;
END_REGION

REGION Network 54: EM Status Enabled
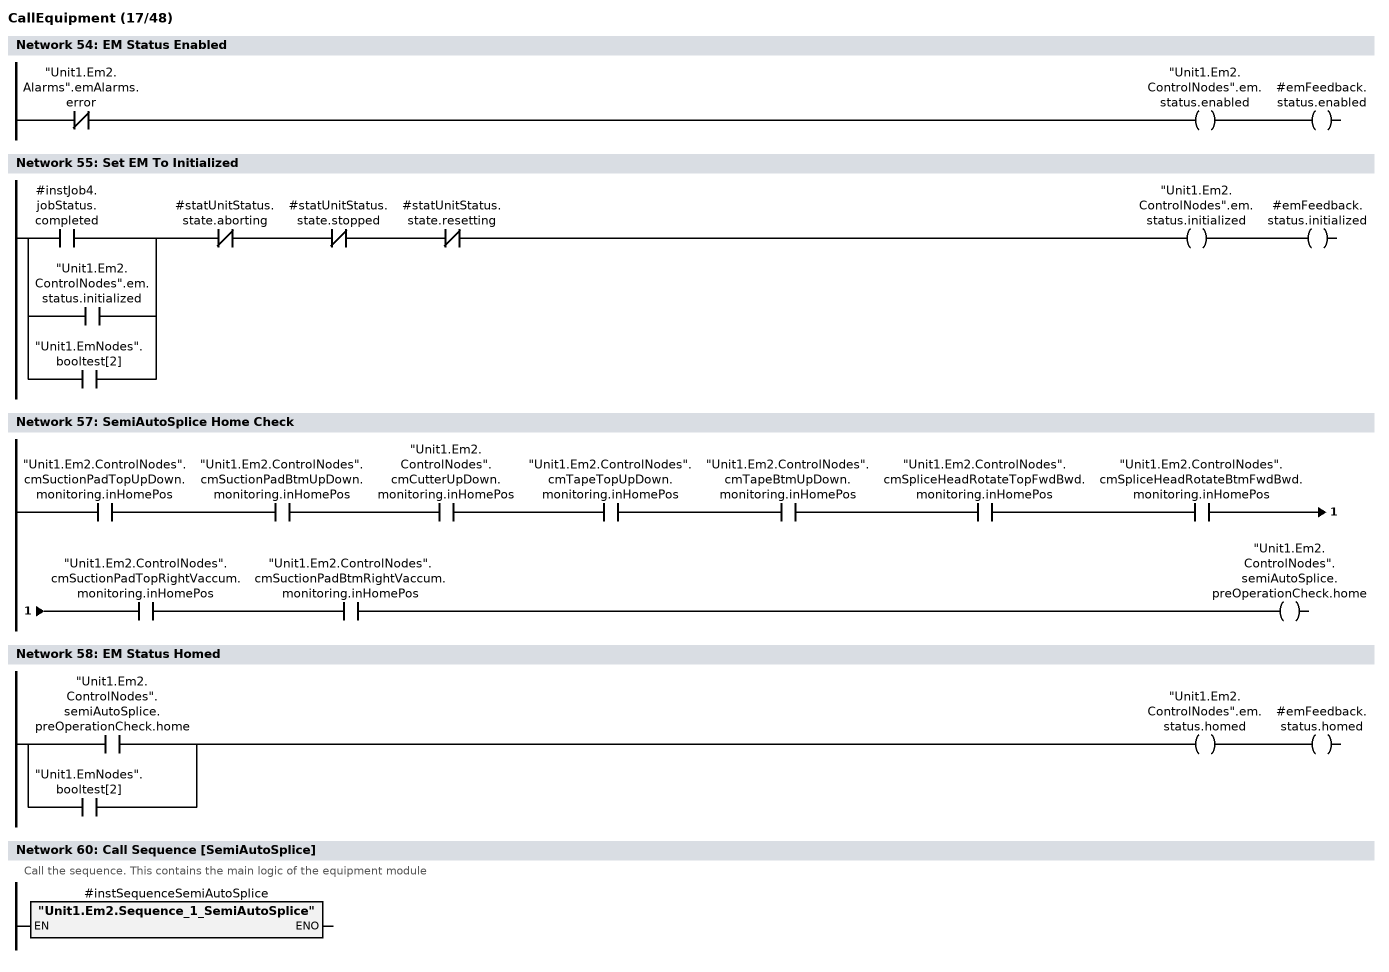
   RUNG wire#powerrail
      I_Contact( "Unit1.Em2.Alarms".emAlarms.error )
      Coil( "Unit1.Em2.ControlNodes".em.status.enabled )
      Coil( #emFeedback.status.enabled )
   END_RUNG
   // the same network as SCL:
   "Unit1.Em2.ControlNodes".em.status.enabled := NOT "Unit1.Em2.Alarms".emAlarms.error;
   #emFeedback.status.enabled := NOT "Unit1.Em2.Alarms".emAlarms.error;
END_REGION

REGION Network 55: Set EM To Initialized
   RUNG wire#powerrail
      Contact( #instJob4.jobStatus.completed )
      wire#w1
      I_Contact( #statUnitStatus.state.aborting )
      I_Contact( #statUnitStatus.state.stopped )
      I_Contact( #statUnitStatus.state.resetting )
      Coil( "Unit1.Em2.ControlNodes".em.status.initialized )
      Coil( #emFeedback.status.initialized )
   END_RUNG
   RUNG wire#powerrail
      Contact( "Unit1.Em2.ControlNodes".em.status.initialized )
   END_RUNG wire#w1
   RUNG wire#powerrail
      Contact( "Unit1.EmNodes".booltest[2] )
   END_RUNG wire#w1
   // the same network as SCL:
   "Unit1.Em2.ControlNodes".em.status.initialized := (#instJob4.jobStatus.completed OR "Unit1.Em2.ControlNodes".em.status.initialized OR "Unit1.EmNodes".booltest[2]) AND NOT #statUnitStatus.state.aborting AND NOT #statUnitStatus.state.stopped AND NOT #statUnitStatus.state.resetting;
   #emFeedback.status.initialized := "Unit1.Em2.ControlNodes".em.status.initialized;
END_REGION

REGION Network 57: SemiAutoSplice Home Check
   RUNG wire#powerrail
      Contact( "Unit1.Em2.ControlNodes".cmSuctionPadTopUpDown.monitoring.inHomePos )
      Contact( "Unit1.Em2.ControlNodes".cmSuctionPadBtmUpDown.monitoring.inHomePos )
      Contact( "Unit1.Em2.ControlNodes".cmCutterUpDown.monitoring.inHomePos )
      Contact( "Unit1.Em2.ControlNodes".cmTapeTopUpDown.monitoring.inHomePos )
      Contact( "Unit1.Em2.ControlNodes".cmTapeBtmUpDown.monitoring.inHomePos )
      Contact( "Unit1.Em2.ControlNodes".cmSpliceHeadRotateTopFwdBwd.monitoring.inHomePos )
      Contact( "Unit1.Em2.ControlNodes".cmSpliceHeadRotateBtmFwdBwd.monitoring.inHomePos )
      Contact( "Unit1.Em2.ControlNodes".cmSuctionPadTopRightVaccum.monitoring.inHomePos )
      Contact( "Unit1.Em2.ControlNodes".cmSuctionPadBtmRightVaccum.monitoring.inHomePos )
      Coil( "Unit1.Em2.ControlNodes".semiAutoSplice.preOperationCheck.home )
   END_RUNG
   // the same network as SCL:
   "Unit1.Em2.ControlNodes".semiAutoSplice.preOperationCheck.home := "Unit1.Em2.ControlNodes".cmSuctionPadTopUpDown.monitoring.inHomePos AND "Unit1.Em2.ControlNodes".cmSuctionPadBtmUpDown.monitoring.inHomePos AND "Unit1.Em2.ControlNodes".cmCutterUpDown.monitoring.inHomePos AND "Unit1.Em2.ControlNodes".cmTapeTopUpDown.monitoring.inHomePos AND "Unit1.Em2.ControlNodes".cmTapeBtmUpDown.monitoring.inHomePos AND "Unit1.Em2.ControlNodes".cmSpliceHeadRotateTopFwdBwd.monitoring.inHomePos AND "Unit1.Em2.ControlNodes".cmSpliceHeadRotateBtmFwdBwd.monitoring.inHomePos AND "Unit1.Em2.ControlNodes".cmSuctionPadTopRightVaccum.monitoring.inHomePos AND "Unit1.Em2.ControlNodes".cmSuctionPadBtmRightVaccum.monitoring.inHomePos;
END_REGION

REGION Network 58: EM Status Homed
   RUNG wire#powerrail
      Contact( "Unit1.Em2.ControlNodes".semiAutoSplice.preOperationCheck.home )
      wire#w1
      Coil( "Unit1.Em2.ControlNodes".em.status.homed )
      Coil( #emFeedback.status.homed )
   END_RUNG
   RUNG wire#powerrail
      Contact( "Unit1.EmNodes".booltest[2] )
   END_RUNG wire#w1
   // the same network as SCL:
   "Unit1.Em2.ControlNodes".em.status.homed := "Unit1.Em2.ControlNodes".semiAutoSplice.preOperationCheck.home OR "Unit1.EmNodes".booltest[2];
   #emFeedback.status.homed := "Unit1.Em2.ControlNodes".em.status.homed;
END_REGION

REGION Network 60: Call Sequence [SemiAutoSplice]
   // Call the sequence. This contains the main logic of the equipment module
   RUNG wire#powerrail
      #instSequenceSemiAutoSplice()
   END_RUNG
   // the same network as SCL:
   #instSequenceSemiAutoSplice();   // "Unit1.Em2.Sequence_1_SemiAutoSplice"
END_REGION

REGION Network 62: ********** Control Modules (TwoWayActuator) **********
   // Call control modules that are actuators after the em logic (jobs and sequence), so that the latest commands are applied to the actuators.
END_REGION

